KUKA KRL program: makrostep9.src

&ACCESS RVO
&COMMENT MakroStep9-Basic
&PARAM TEMPLATE = C:\KRC\Roboter\Template\makrostepvorgabe.src
&PARAM EDITMASK = MakroStep
&PARAM TPVW_VERSION = 8.3.15
DEF MAKROSTEP9(Function :IN)
   ; FOLD Makro Schrittkette;%{SE} %MKUKATPVW
   ; FOLD ;%{H} %MKUKATPVW
   INT Function
   IF Function==1 THEN
     APP_INT_STEP[9]=1
     Return
   ENDIF
   SWITCH APP_INT_STEP[9]
   Case 0
   ; ENDFOLD
   ;ENDFOLD
   ;FOLD SCHRITT 1 -- -- ;%{P}%MKUKATPVW,%CSTEP,%VST_NR,%P 1:SCHRITT, 2:1, 3:
      ;FOLD ;%{H}
         Case 1
      ;ENDFOLD
      ;FOLD -- Roboter Schrittkette -- ;%{SE}%MKUKATPVW %CVW_COM %VCOMMENT %P 2:-- Roboter Schrittkette --, 3: VW_COMMENT
      ;ENDFOLD
      ;FOLD -- KS26 -- ;%{SE}%MKUKATPVW %CVW_COM %VCOMMENT %P 2:-- KS26 --, 3: VW_COMMENT
      ;ENDFOLD
      ;FOLD -- Version: 01 -- ;%{SE}%MKUKATPVW %CVW_COM %VCOMMENT %P 2:-- Version: 01 --, 3: VW_COMMENT
      ;ENDFOLD
      ;FOLD -- Stand: 008 -- ;%{SE}%MKUKATPVW %CVW_COM %VCOMMENT %P 2:-- Stand: 008 --, 3: VW_COMMENT
      ;ENDFOLD
      ;FOLD -- letzte Aenderung 11.07.2019 LZ -- ;%{SE}%MKUKATPVW %CVW_COM %VCOMMENT %P 2:-- letzte Aenderung 11.07.2019 LZ --, 3: VW_COMMENT
      ;ENDFOLD
      ;FOLD -- E/A's und Flags Ruecksetzen -- ;%{SE}%MKUKATPVW %CVW_COM %VCOMMENT %P 2:-- E/A's und Flags Ruecksetzen --, 3: VW_COMMENT
      ;ENDFOLD
      ;FOLD -- SK1 KF1 KS1 KE1 -- ;%{SE}%MKUKATPVW %CVW_COM %VCOMMENT %P 2:-- SK1 KF1 KS1 KE1 --, 3: VW_COMMENT
      ;ENDFOLD
      ;FOLD A786 = F830 & A786 ;%{SE}%MKUKATPVW %CVW_SPS %VBOASG %P 2:A786 = F830 & A786, 3: BOASG
         $OUT[786] = $FLAG[830] AND $OUT[786]
      ;ENDFOLD
      ;FOLD A722 = !F830 & A722 ;%{SE}%MKUKATPVW %CVW_SPS %VBOASG %P 2:A722 = !F830 & A722, 3: BOASG
         $OUT[722] = NOT $FLAG[830] AND $OUT[722]
      ;ENDFOLD
      ;FOLD A834 = AUS ;%{SE}%MKUKATPVW %CVW_SPS %VBOASG %P 2:A834 = AUS, 3: BOASG
         $OUT[834] = FALSE
      ;ENDFOLD
      ;FOLD A840 = AUS ;%{SE}%MKUKATPVW %CVW_SPS %VBOASG %P 2:A840 = AUS, 3: BOASG
         $OUT[840] = FALSE
      ;ENDFOLD
      ;FOLD A757 = AUS ;%{SE}%MKUKATPVW %CVW_SPS %VBOASG %P 2:A757 = AUS, 3: BOASG
         $OUT[757] = FALSE
      ;ENDFOLD
      ;FOLD -- SK2 KF2 KS2 KE2 -- ;%{SE}%MKUKATPVW %CVW_COM %VCOMMENT %P 2:-- SK2 KF2 KS2 KE2 --, 3: VW_COMMENT
      ;ENDFOLD
      ;FOLD A946 = F831 & A946 ;%{SE}%MKUKATPVW %CVW_SPS %VBOASG %P 2:A946 = F831 & A946, 3: BOASG
         $OUT[946] = $FLAG[831] AND $OUT[946]
      ;ENDFOLD
      ;FOLD A882 = !F831 & A882 ;%{SE}%MKUKATPVW %CVW_SPS %VBOASG %P 2:A882 = !F831 & A882, 3: BOASG
         $OUT[882] = NOT $FLAG[831] AND $OUT[882]
      ;ENDFOLD
      ;FOLD A994 = AUS ;%{SE}%MKUKATPVW %CVW_SPS %VBOASG %P 2:A994 = AUS, 3: BOASG
         $OUT[994] = FALSE
      ;ENDFOLD
      ;FOLD A995 = AUS ;%{SE}%MKUKATPVW %CVW_SPS %VBOASG %P 2:A995 = AUS, 3: BOASG
         $OUT[995] = FALSE
      ;ENDFOLD
      ;FOLD A1000 = AUS ;%{SE}%MKUKATPVW %CVW_SPS %VBOASG %P 2:A1000 = AUS, 3: BOASG
         $OUT[1000] = FALSE
      ;ENDFOLD
      ;FOLD -- SK3 KF3 KS3 KE3 -- ;%{SE}%MKUKATPVW %CVW_COM %VCOMMENT %P 2:-- SK3 KF3 KS3 KE3 --, 3: VW_COMMENT
      ;ENDFOLD
      ;FOLD A1106 = F832 & A1106 ;%{SE}%MKUKATPVW %CVW_SPS %VBOASG %P 2:A1106 = F832 & A1106, 3: BOASG
         $OUT[1106] = $FLAG[832] AND $OUT[1106]
      ;ENDFOLD
      ;FOLD A1042 = !F832 & A1042 ;%{SE}%MKUKATPVW %CVW_SPS %VBOASG %P 2:A1042 = !F832 & A1042, 3: BOASG
         $OUT[1042] = NOT $FLAG[832] AND $OUT[1042]
      ;ENDFOLD
      ;FOLD A1154 = AUS ;%{SE}%MKUKATPVW %CVW_SPS %VBOASG %P 2:A1154 = AUS, 3: BOASG
         $OUT[1154] = FALSE
      ;ENDFOLD
      ;FOLD A1155 = AUS ;%{SE}%MKUKATPVW %CVW_SPS %VBOASG %P 2:A1155 = AUS, 3: BOASG
         $OUT[1155] = FALSE
      ;ENDFOLD
      ;FOLD A1160 = AUS ;%{SE}%MKUKATPVW %CVW_SPS %VBOASG %P 2:A1160 = AUS, 3: BOASG
         $OUT[1160] = FALSE
      ;ENDFOLD
      ;FOLD -- Auswertung KF Umdrehungen ServoGun -- ;%{SE}%MKUKATPVW %CVW_COM %VCOMMENT %P 2:-- Auswertung KF Umdrehungen ServoGun --, 3: VW_COMMENT
      ;ENDFOLD
      ;FOLD F94 = AUS ;%{SE}%MKUKATPVW %CVW_SPS %VBOASG %P 2:F94 = AUS, 3: BOASG
         $FLAG[94] = FALSE
      ;ENDFOLD
      ;FOLD F95 = AUS ;%{SE}%MKUKATPVW %CVW_SPS %VBOASG %P 2:F95 = AUS, 3: BOASG
         $FLAG[95] = FALSE
      ;ENDFOLD
      ;FOLD F96 = AUS ;%{SE}%MKUKATPVW %CVW_SPS %VBOASG %P 2:F96 = AUS, 3: BOASG
         $FLAG[96] = FALSE
      ;ENDFOLD
      ;FOLD F97 = AUS ;%{SE}%MKUKATPVW %CVW_SPS %VBOASG %P 2:F97 = AUS, 3: BOASG
         $FLAG[97] = FALSE
      ;ENDFOLD
      ;FOLD F98 = AUS ;%{SE}%MKUKATPVW %CVW_SPS %VBOASG %P 2:F98 = AUS, 3: BOASG
         $FLAG[98] = FALSE
      ;ENDFOLD
      ;FOLD F99 = AUS ;%{SE}%MKUKATPVW %CVW_SPS %VBOASG %P 2:F99 = AUS, 3: BOASG
         $FLAG[99] = FALSE
      ;ENDFOLD
      ;FOLD F100 = AUS ;%{SE}%MKUKATPVW %CVW_SPS %VBOASG %P 2:F100 = AUS, 3: BOASG
         $FLAG[100] = FALSE
      ;ENDFOLD
      ;FOLD F101 = AUS ;%{SE}%MKUKATPVW %CVW_SPS %VBOASG %P 2:F101 = AUS, 3: BOASG
         $FLAG[101] = FALSE
      ;ENDFOLD
      ;FOLD F102 = AUS ;%{SE}%MKUKATPVW %CVW_SPS %VBOASG %P 2:F102 = AUS, 3: BOASG
         $FLAG[102] = FALSE
      ;ENDFOLD
      ;FOLD F103 = AUS ;%{SE}%MKUKATPVW %CVW_SPS %VBOASG %P 2:F103 = AUS, 3: BOASG
         $FLAG[103] = FALSE
      ;ENDFOLD
      ;FOLD F104 = AUS ;%{SE}%MKUKATPVW %CVW_SPS %VBOASG %P 2:F104 = AUS, 3: BOASG
         $FLAG[104] = FALSE
      ;ENDFOLD
      ;FOLD F105 = AUS ;%{SE}%MKUKATPVW %CVW_SPS %VBOASG %P 2:F105 = AUS, 3: BOASG
         $FLAG[105] = FALSE
      ;ENDFOLD
      ;FOLD F106 = AUS ;%{SE}%MKUKATPVW %CVW_SPS %VBOASG %P 2:F106 = AUS, 3: BOASG
         $FLAG[106] = FALSE
      ;ENDFOLD
      ;FOLD F107 = AUS ;%{SE}%MKUKATPVW %CVW_SPS %VBOASG %P 2:F107 = AUS, 3: BOASG
         $FLAG[107] = FALSE
      ;ENDFOLD
      ;FOLD F108 = AUS ;%{SE}%MKUKATPVW %CVW_SPS %VBOASG %P 2:F108 = AUS, 3: BOASG
         $FLAG[108] = FALSE
      ;ENDFOLD
      ;FOLD F109 = AUS ;%{SE}%MKUKATPVW %CVW_SPS %VBOASG %P 2:F109 = AUS, 3: BOASG
         $FLAG[109] = FALSE
      ;ENDFOLD
      ;FOLD F110 = AUS ;%{SE}%MKUKATPVW %CVW_SPS %VBOASG %P 2:F110 = AUS, 3: BOASG
         $FLAG[110] = FALSE
      ;ENDFOLD
      ;FOLD F111 = AUS ;%{SE}%MKUKATPVW %CVW_SPS %VBOASG %P 2:F111 = AUS, 3: BOASG
         $FLAG[111] = FALSE
      ;ENDFOLD
      ;FOLD F112 = AUS ;%{SE}%MKUKATPVW %CVW_SPS %VBOASG %P 2:F112 = AUS, 3: BOASG
         $FLAG[112] = FALSE
      ;ENDFOLD
      ;FOLD F113 = AUS ;%{SE}%MKUKATPVW %CVW_SPS %VBOASG %P 2:F113 = AUS, 3: BOASG
         $FLAG[113] = FALSE
      ;ENDFOLD
      ;FOLD F114 = AUS ;%{SE}%MKUKATPVW %CVW_SPS %VBOASG %P 2:F114 = AUS, 3: BOASG
         $FLAG[114] = FALSE
      ;ENDFOLD
      ;FOLD F115 = AUS ;%{SE}%MKUKATPVW %CVW_SPS %VBOASG %P 2:F115 = AUS, 3: BOASG
         $FLAG[115] = FALSE
      ;ENDFOLD
      ;FOLD F116 = AUS ;%{SE}%MKUKATPVW %CVW_SPS %VBOASG %P 2:F116 = AUS, 3: BOASG
         $FLAG[116] = FALSE
      ;ENDFOLD
      ;FOLD F117 = AUS ;%{SE}%MKUKATPVW %CVW_SPS %VBOASG %P 2:F117 = AUS, 3: BOASG
         $FLAG[117] = FALSE
      ;ENDFOLD
      ;FOLD -- Auswertung KF Umdrehungen EZ2/SP2/KE2 -- ;%{SE}%MKUKATPVW %CVW_COM %VCOMMENT %P 2:-- Auswertung KF Umdrehungen EZ2/SP2/KE2 --, 3: VW_COMMENT
      ;ENDFOLD
      ;FOLD F150 = AUS ;%{SE}%MKUKATPVW %CVW_SPS %VBOASG %P 2:F150 = AUS, 3: BOASG
         $FLAG[150] = FALSE
      ;ENDFOLD
      ;FOLD F151 = AUS ;%{SE}%MKUKATPVW %CVW_SPS %VBOASG %P 2:F151 = AUS, 3: BOASG
         $FLAG[151] = FALSE
      ;ENDFOLD
      ;FOLD F152 = AUS ;%{SE}%MKUKATPVW %CVW_SPS %VBOASG %P 2:F152 = AUS, 3: BOASG
         $FLAG[152] = FALSE
      ;ENDFOLD
      ;FOLD F153 = AUS ;%{SE}%MKUKATPVW %CVW_SPS %VBOASG %P 2:F153 = AUS, 3: BOASG
         $FLAG[153] = FALSE
      ;ENDFOLD
      ;FOLD F154 = AUS ;%{SE}%MKUKATPVW %CVW_SPS %VBOASG %P 2:F154 = AUS, 3: BOASG
         $FLAG[154] = FALSE
      ;ENDFOLD
      ;FOLD F155 = AUS ;%{SE}%MKUKATPVW %CVW_SPS %VBOASG %P 2:F155 = AUS, 3: BOASG
         $FLAG[155] = FALSE
      ;ENDFOLD
      ;FOLD -- Auswertung KF Umdrehungen EZ3/SP3/KE3 -- ;%{SE}%MKUKATPVW %CVW_COM %VCOMMENT %P 2:-- Auswertung KF Umdrehungen EZ3/SP3/KE3 --, 3: VW_COMMENT
      ;ENDFOLD
      ;FOLD F186 = AUS ;%{SE}%MKUKATPVW %CVW_SPS %VBOASG %P 2:F186 = AUS, 3: BOASG
         $FLAG[186] = FALSE
      ;ENDFOLD
      ;FOLD F187 = AUS ;%{SE}%MKUKATPVW %CVW_SPS %VBOASG %P 2:F187 = AUS, 3: BOASG
         $FLAG[187] = FALSE
      ;ENDFOLD
      ;FOLD F188 = AUS ;%{SE}%MKUKATPVW %CVW_SPS %VBOASG %P 2:F188 = AUS, 3: BOASG
         $FLAG[188] = FALSE
      ;ENDFOLD
      ;FOLD F189 = AUS ;%{SE}%MKUKATPVW %CVW_SPS %VBOASG %P 2:F189 = AUS, 3: BOASG
         $FLAG[189] = FALSE
      ;ENDFOLD
      ;FOLD F190 = AUS ;%{SE}%MKUKATPVW %CVW_SPS %VBOASG %P 2:F190 = AUS, 3: BOASG
         $FLAG[190] = FALSE
      ;ENDFOLD
      ;FOLD F191 = AUS ;%{SE}%MKUKATPVW %CVW_SPS %VBOASG %P 2:F191 = AUS, 3: BOASG
         $FLAG[191] = FALSE
      ;ENDFOLD
      ;FOLD -- Hilfsflags beim Fraesen -- ;%{SE}%MKUKATPVW %CVW_COM %VCOMMENT %P 2:-- Hilfsflags beim Fraesen --, 3: VW_COMMENT
      ;ENDFOLD
      ;FOLD F749 = AUS ;%{SE}%MKUKATPVW %CVW_SPS %VBOASG %P 2:F749 = AUS, 3: BOASG
         $FLAG[749] = FALSE
      ;ENDFOLD
      ;FOLD F287 = AUS ;%{SE}%MKUKATPVW %CVW_SPS %VBOASG %P 2:F287 = AUS, 3: BOASG
         $FLAG[287] = FALSE
      ;ENDFOLD
      ;FOLD F290 = AUS ;%{SE}%MKUKATPVW %CVW_SPS %VBOASG %P 2:F290 = AUS, 3: BOASG
         $FLAG[290] = FALSE
      ;ENDFOLD
      ;FOLD F291 = AUS ;%{SE}%MKUKATPVW %CVW_SPS %VBOASG %P 2:F291 = AUS, 3: BOASG
         $FLAG[291] = FALSE
      ;ENDFOLD
      ;FOLD -- Hilfsflags SZ2 an SK1 -- ;%{SE}%MKUKATPVW %CVW_COM %VCOMMENT %P 2:-- Hilfsflags SZ2 an SK1 --, 3: VW_COMMENT
      ;ENDFOLD
      ;FOLD F307 = AUS ;%{SE}%MKUKATPVW %CVW_SPS %VBOASG %P 2:F307 = AUS, 3: BOASG
         $FLAG[307] = FALSE
      ;ENDFOLD
      ;FOLD F308 = AUS ;%{SE}%MKUKATPVW %CVW_SPS %VBOASG %P 2:F308 = AUS, 3: BOASG
         $FLAG[308] = FALSE
      ;ENDFOLD
      ;FOLD -- Hilfsflags Funktionstest KF Motor -- ;%{SE}%MKUKATPVW %CVW_COM %VCOMMENT %P 2:-- Hilfsflags Funktionstest KF Motor --, 3: VW_COMMENT
      ;ENDFOLD
      ;FOLD F312 = AUS ;%{SE}%MKUKATPVW %CVW_SPS %VBOASG %P 2:F312 = AUS, 3: BOASG
         $FLAG[312] = FALSE
      ;ENDFOLD
      ;FOLD F313 = AUS ;%{SE}%MKUKATPVW %CVW_SPS %VBOASG %P 2:F313 = AUS, 3: BOASG
         $FLAG[313] = FALSE
      ;ENDFOLD
      ;FOLD -- RSK Fehlerausgaben -- ;%{SE}%MKUKATPVW %CVW_COM %VCOMMENT %P 2:-- RSK Fehlerausgaben --, 3: VW_COMMENT
      ;ENDFOLD
      ;FOLD F322 = AUS ;%{SE}%MKUKATPVW %CVW_SPS %VBOASG %P 2:F322 = AUS, 3: BOASG
         $FLAG[322] = FALSE
      ;ENDFOLD
      ;FOLD F323 = AUS ;%{SE}%MKUKATPVW %CVW_SPS %VBOASG %P 2:F323 = AUS, 3: BOASG
         $FLAG[323] = FALSE
      ;ENDFOLD
      ;FOLD F324 = AUS ;%{SE}%MKUKATPVW %CVW_SPS %VBOASG %P 2:F324 = AUS, 3: BOASG
         $FLAG[324] = FALSE
      ;ENDFOLD
      ;FOLD F325 = AUS ;%{SE}%MKUKATPVW %CVW_SPS %VBOASG %P 2:F325 = AUS, 3: BOASG
         $FLAG[325] = FALSE
      ;ENDFOLD
      ;FOLD F326 = AUS ;%{SE}%MKUKATPVW %CVW_SPS %VBOASG %P 2:F326 = AUS, 3: BOASG
         $FLAG[326] = FALSE
      ;ENDFOLD
      ;FOLD F327 = AUS ;%{SE}%MKUKATPVW %CVW_SPS %VBOASG %P 2:F327 = AUS, 3: BOASG
         $FLAG[327] = FALSE
      ;ENDFOLD
      ;FOLD F328 = AUS ;%{SE}%MKUKATPVW %CVW_SPS %VBOASG %P 2:F328 = AUS, 3: BOASG
         $FLAG[328] = FALSE
      ;ENDFOLD
      ;FOLD F329 = AUS ;%{SE}%MKUKATPVW %CVW_SPS %VBOASG %P 2:F329 = AUS, 3: BOASG
         $FLAG[329] = FALSE
      ;ENDFOLD
      ;FOLD A3518 = AUS ;%{SE}%MKUKATPVW %CVW_SPS %VBOASG %P 2:A3518 = AUS, 3: BOASG
         $OUT[3518] = FALSE
      ;ENDFOLD
      ;FOLD A3519 = AUS ;%{SE}%MKUKATPVW %CVW_SPS %VBOASG %P 2:A3519 = AUS, 3: BOASG
         $OUT[3519] = FALSE
      ;ENDFOLD
      ;FOLD -- Schritt Fraesen aktiv -- ;%{SE}%MKUKATPVW %CVW_COM %VCOMMENT %P 2:-- Schritt Fraesen aktiv --, 3: VW_COMMENT
      ;ENDFOLD
      ;FOLD A3534 = AUS ;%{SE}%MKUKATPVW %CVW_SPS %VBOASG %P 2:A3534 = AUS, 3: BOASG
         $OUT[3534] = FALSE
      ;ENDFOLD
      ;FOLD -- Schritt Messen aktiv -- ;%{SE}%MKUKATPVW %CVW_COM %VCOMMENT %P 2:-- Schritt Messen aktiv --, 3: VW_COMMENT
      ;ENDFOLD
      ;FOLD A3535 = AUS ;%{SE}%MKUKATPVW %CVW_SPS %VBOASG %P 2:A3535 = AUS, 3: BOASG
         $OUT[3535] = FALSE
      ;ENDFOLD
      ;FOLD -- Schritt Schweissen aktiv -- ;%{SE}%MKUKATPVW %CVW_COM %VCOMMENT %P 2:-- Schritt Schweissen aktiv --, 3: VW_COMMENT
      ;ENDFOLD
      ;FOLD A3536 = AUS ;%{SE}%MKUKATPVW %CVW_SPS %VBOASG %P 2:A3536 = AUS, 3: BOASG
         $OUT[3536] = FALSE
      ;ENDFOLD
      ;FOLD -- Hilfsflag SK Programmwechsel -- ;%{SE}%MKUKATPVW %CVW_COM %VCOMMENT %P 2:-- Hilfsflag SK Programmwechsel --, 3: VW_COMMENT
      ;ENDFOLD
      ;FOLD F334 = AUS ;%{SE}%MKUKATPVW %CVW_SPS %VBOASG %P 2:F334 = AUS, 3: BOASG
         $FLAG[334] = FALSE
      ;ENDFOLD
      ;FOLD -- Timer Stoppen -- ;%{SE}%MKUKATPVW %CVW_COM %VCOMMENT %P 2:-- Timer Stoppen --, 3: VW_COMMENT
      ;ENDFOLD
      ;FOLD t7 ( EIN ) = STOP ;%{SE}%MKUKATPVW %CVW_SPS %VTSTOP %P 2:t7 ( EIN ) = STOP, 3: TSTOP
         VW(#SET_TIME,TRUE,7,1,0)
      ;ENDFOLD
      ;FOLD t8 ( EIN ) = STOP ;%{SE}%MKUKATPVW %CVW_SPS %VTSTOP %P 2:t8 ( EIN ) = STOP, 3: TSTOP
         VW(#SET_TIME,TRUE,8,1,0)
      ;ENDFOLD
      ;FOLD t9 ( EIN ) = STOP ;%{SE}%MKUKATPVW %CVW_SPS %VTSTOP %P 2:t9 ( EIN ) = STOP, 3: TSTOP
         VW(#SET_TIME,TRUE,9,1,0)
      ;ENDFOLD
      ;FOLD Schritt 2 = EIN ;%{SE}%MKUKATPVW %CVW_SPS %VST_CON %P 2:Schritt 2 = EIN, 3: ST_CON
         IF TRUE THEN
            PREV_STEP[9] = APP_INT_STEP[9]
            APP_INT_STEP[9] = 2
         ENDIF
      ;ENDFOLD
   ;ENDFOLD
   ;FOLD SCHRITT 2 --  RSK Grundstellung # Anwahlen-- ;%{P}%MKUKATPVW,%CSTEP,%VST_NR,%P 1:SCHRITT, 2:2, 3:  RSK Grundstellung # Anwahlen
      ;FOLD ;%{H}
         Case 2
      ;ENDFOLD
      ;FOLD -- RSK ServoZange in Grundstellung AUS -- ;%{SE}%MKUKATPVW %CVW_COM %VCOMMENT %P 2:-- RSK ServoZange in Grundstellung AUS --, 3: VW_COMMENT
      ;ENDFOLD
      ;FOLD F276 = AUS ;%{SE}%MKUKATPVW %CVW_SPS %VBOASG %P 2:F276 = AUS, 3: BOASG
         $FLAG[276] = FALSE
      ;ENDFOLD
      ;FOLD -- Fraesen st. RZ Start -- ;%{SE}%MKUKATPVW %CVW_COM %VCOMMENT %P 2:-- Fraesen st. RZ Start --, 3: VW_COMMENT
      ;ENDFOLD
      ;FOLD Schritt 103 = F92 & !F93 & A4039 & E13 & F273 & !F274 & !F275 & !F530 ;%{SE}%MKUKATPVW %CVW_SPS %VST_CON %P 2:Schritt 103 = F92 & !F93 & A4039 & E13 & F273 & !F274 & !F275 & !F530, 3: ST_CON
         IF $FLAG[92] AND NOT $FLAG[93] AND $OUT[4039] AND $IN[13] AND $FLAG[273] AND NOT $FLAG[274] AND NOT $FLAG[275] AND NOT $FLAG[530] THEN
            PREV_STEP[9] = APP_INT_STEP[9]
            APP_INT_STEP[9] = 103
         ENDIF
      ;ENDFOLD
      ;FOLD Schritt 203 = F148 & !F149 & A4039 & E13 & F273 & F274 & !F275  & !F530 ;%{SE}%MKUKATPVW %CVW_SPS %VST_CON %P 2:Schritt 203 = F148 & !F149 & A4039 & E13 & F273 & F274 & !F275  & !F530, 3: ST_CON
         IF $FLAG[148] AND NOT $FLAG[149] AND $OUT[4039] AND $IN[13] AND $FLAG[273] AND $FLAG[274] AND NOT $FLAG[275] AND NOT $FLAG[530] THEN
            PREV_STEP[9] = APP_INT_STEP[9]
            APP_INT_STEP[9] = 203
         ENDIF
      ;ENDFOLD
      ;FOLD Schritt 303 = F184 & !F185 & A4039 & E13 & F273 & F274 & F275  & !F530 ;%{SE}%MKUKATPVW %CVW_SPS %VST_CON %P 2:Schritt 303 = F184 & !F185 & A4039 & E13 & F273 & F274 & F275  & !F530, 3: ST_CON
         IF $FLAG[184] AND NOT $FLAG[185] AND $OUT[4039] AND $IN[13] AND $FLAG[273] AND $FLAG[274] AND $FLAG[275] AND NOT $FLAG[530] THEN
            PREV_STEP[9] = APP_INT_STEP[9]
            APP_INT_STEP[9] = 303
         ENDIF
      ;ENDFOLD
      ;FOLD Schritt 500 = A757 & A4039 & E13 & F273 & F530 ;%{SE}%MKUKATPVW %CVW_SPS %VST_CON %P 2:Schritt 500 = A757 & A4039 & E13 & F273 & F530, 3: ST_CON
         IF $OUT[757] AND $OUT[4039] AND $IN[13] AND $FLAG[273] AND $FLAG[530] THEN
            PREV_STEP[9] = APP_INT_STEP[9]
            APP_INT_STEP[9] = 500
         ENDIF
      ;ENDFOLD
   ;ENDFOLD
   ;FOLD SCHRITT 103 -- st. RZ1 # Start -- ;%{P}%MKUKATPVW,%CSTEP,%VST_NR,%P 1:SCHRITT, 2:103, 3: st. RZ1 # Start
      ;FOLD ;%{H}
         Case 103
      ;ENDFOLD
      ;FOLD -- RSK gestartet -- ;%{SE}%MKUKATPVW %CVW_COM %VCOMMENT %P 2:-- RSK gestartet --, 3: VW_COMMENT
      ;ENDFOLD
      ;FOLD F122 = AUS ;%{SE}%MKUKATPVW %CVW_SPS %VBOASG %P 2:F122 = AUS, 3: BOASG
         $FLAG[122] = FALSE
      ;ENDFOLD
      ;FOLD F322 = AUS ;%{SE}%MKUKATPVW %CVW_SPS %VBOASG %P 2:F322 = AUS, 3: BOASG
         $FLAG[322] = FALSE
      ;ENDFOLD
      ;FOLD F323 = AUS ;%{SE}%MKUKATPVW %CVW_SPS %VBOASG %P 2:F323 = AUS, 3: BOASG
         $FLAG[323] = FALSE
      ;ENDFOLD
      ;FOLD F324 = AUS ;%{SE}%MKUKATPVW %CVW_SPS %VBOASG %P 2:F324 = AUS, 3: BOASG
         $FLAG[324] = FALSE
      ;ENDFOLD
      ;FOLD F325 = AUS ;%{SE}%MKUKATPVW %CVW_SPS %VBOASG %P 2:F325 = AUS, 3: BOASG
         $FLAG[325] = FALSE
      ;ENDFOLD
      ;FOLD F326 = AUS ;%{SE}%MKUKATPVW %CVW_SPS %VBOASG %P 2:F326 = AUS, 3: BOASG
         $FLAG[326] = FALSE
      ;ENDFOLD
      ;FOLD F327 = AUS ;%{SE}%MKUKATPVW %CVW_SPS %VBOASG %P 2:F327 = AUS, 3: BOASG
         $FLAG[327] = FALSE
      ;ENDFOLD
      ;FOLD F329 = AUS ;%{SE}%MKUKATPVW %CVW_SPS %VBOASG %P 2:F329 = AUS, 3: BOASG
         $FLAG[329] = FALSE
      ;ENDFOLD
      ;FOLD -- ServoGun SZ1 Zaehler -- ;%{SE}%MKUKATPVW %CVW_COM %VCOMMENT %P 2:-- ServoGun SZ1 Zaehler --, 3: VW_COMMENT
      ;ENDFOLD
      ;FOLD F94 = AUS ;%{SE}%MKUKATPVW %CVW_SPS %VBOASG %P 2:F94 = AUS, 3: BOASG
         $FLAG[94] = FALSE
      ;ENDFOLD
      ;FOLD F95 = AUS ;%{SE}%MKUKATPVW %CVW_SPS %VBOASG %P 2:F95 = AUS, 3: BOASG
         $FLAG[95] = FALSE
      ;ENDFOLD
      ;FOLD F96 = AUS ;%{SE}%MKUKATPVW %CVW_SPS %VBOASG %P 2:F96 = AUS, 3: BOASG
         $FLAG[96] = FALSE
      ;ENDFOLD
      ;FOLD F97 = AUS ;%{SE}%MKUKATPVW %CVW_SPS %VBOASG %P 2:F97 = AUS, 3: BOASG
         $FLAG[97] = FALSE
      ;ENDFOLD
      ;FOLD F98 = AUS ;%{SE}%MKUKATPVW %CVW_SPS %VBOASG %P 2:F98 = AUS, 3: BOASG
         $FLAG[98] = FALSE
      ;ENDFOLD
      ;FOLD F99 = AUS ;%{SE}%MKUKATPVW %CVW_SPS %VBOASG %P 2:F99 = AUS, 3: BOASG
         $FLAG[99] = FALSE
      ;ENDFOLD
      ;FOLD -- Hilfsflags Funktionstest KF Motor -- ;%{SE}%MKUKATPVW %CVW_COM %VCOMMENT %P 2:-- Hilfsflags Funktionstest KF Motor --, 3: VW_COMMENT
      ;ENDFOLD
      ;FOLD F312 = AUS ;%{SE}%MKUKATPVW %CVW_SPS %VBOASG %P 2:F312 = AUS, 3: BOASG
         $FLAG[312] = FALSE
      ;ENDFOLD
      ;FOLD F313 = AUS ;%{SE}%MKUKATPVW %CVW_SPS %VBOASG %P 2:F313 = AUS, 3: BOASG
         $FLAG[313] = FALSE
      ;ENDFOLD
      ;FOLD -- Hilfsflags ServoGun Start -- ;%{SE}%MKUKATPVW %CVW_COM %VCOMMENT %P 2:-- Hilfsflags ServoGun Start --, 3: VW_COMMENT
      ;ENDFOLD
      ;FOLD F276 = EIN ;%{SE}%MKUKATPVW %CVW_SPS %VBOASG %P 2:F276 = EIN, 3: BOASG
         $FLAG[276] = TRUE
      ;ENDFOLD
      ;FOLD A3871 = AUS ;%{SE}%MKUKATPVW %CVW_SPS %VBOASG %P 2:A3871 = AUS, 3: BOASG
         $OUT[3871] = FALSE
      ;ENDFOLD
      ;FOLD A3872 = AUS ;%{SE}%MKUKATPVW %CVW_SPS %VBOASG %P 2:A3872 = AUS, 3: BOASG
         $OUT[3872] = FALSE
      ;ENDFOLD
      ;FOLD A3510 = EIN ;%{SE}%MKUKATPVW %CVW_SPS %VBOASG %P 2:A3510 = EIN, 3: BOASG
         $OUT[3510] = TRUE
      ;ENDFOLD
      ;FOLD A3511 = AUS ;%{SE}%MKUKATPVW %CVW_SPS %VBOASG %P 2:A3511 = AUS, 3: BOASG
         $OUT[3511] = FALSE
      ;ENDFOLD
      ;FOLD A3514 = AUS ;%{SE}%MKUKATPVW %CVW_SPS %VBOASG %P 2:A3514 = AUS, 3: BOASG
         $OUT[3514] = FALSE
      ;ENDFOLD
      ;FOLD A3513 = AUS ;%{SE}%MKUKATPVW %CVW_SPS %VBOASG %P 2:A3513 = AUS, 3: BOASG
         $OUT[3513] = FALSE
      ;ENDFOLD
      ;FOLD A3512 = AUS ;%{SE}%MKUKATPVW %CVW_SPS %VBOASG %P 2:A3512 = AUS, 3: BOASG
         $OUT[3512] = FALSE
      ;ENDFOLD
      ;FOLD A3533 = AUS ;%{SE}%MKUKATPVW %CVW_SPS %VBOASG %P 2:A3533 = AUS, 3: BOASG
         $OUT[3533] = FALSE
      ;ENDFOLD
      ;FOLD A3534 = AUS ;%{SE}%MKUKATPVW %CVW_SPS %VBOASG %P 2:A3534 = AUS, 3: BOASG
         $OUT[3534] = FALSE
      ;ENDFOLD
      ;FOLD A3535 = AUS ;%{SE}%MKUKATPVW %CVW_SPS %VBOASG %P 2:A3535 = AUS, 3: BOASG
         $OUT[3535] = FALSE
      ;ENDFOLD
      ;FOLD A3536 = AUS ;%{SE}%MKUKATPVW %CVW_SPS %VBOASG %P 2:A3536 = AUS, 3: BOASG
         $OUT[3536] = FALSE
      ;ENDFOLD
      ;FOLD -- Hilfsflags ServoGun Ende -- ;%{SE}%MKUKATPVW %CVW_COM %VCOMMENT %P 2:-- Hilfsflags ServoGun Ende --, 3: VW_COMMENT
      ;ENDFOLD
      ;FOLD -- Ausblasen zuruecksetzen -- ;%{SE}%MKUKATPVW %CVW_COM %VCOMMENT %P 2:-- Ausblasen zuruecksetzen --, 3: VW_COMMENT
      ;ENDFOLD
      ;FOLD A836 = AUS ;%{SE}%MKUKATPVW %CVW_SPS %VBOASG %P 2:A836 = AUS, 3: BOASG
         $OUT[836] = FALSE
      ;ENDFOLD
      ;FOLD A996 = AUS ;%{SE}%MKUKATPVW %CVW_SPS %VBOASG %P 2:A996 = AUS, 3: BOASG
         $OUT[996] = FALSE
      ;ENDFOLD
      ;FOLD A1156 = AUS ;%{SE}%MKUKATPVW %CVW_SPS %VBOASG %P 2:A1156 = AUS, 3: BOASG
         $OUT[1156] = FALSE
      ;ENDFOLD
      ;FOLD -- Prognummer setzen -- ;%{SE}%MKUKATPVW %CVW_COM %VCOMMENT %P 2:-- Prognummer setzen --, 3: VW_COMMENT
      ;ENDFOLD
      ;FOLD bin28 ( EIN ) = 0 ;%{SE}%MKUKATPVW %CVW_SPS %VARIASG %P 2:bin28 ( EIN ) = 0, 3: ARIASG
         VW(#BINOUT,TRUE,28,0)
      ;ENDFOLD
      ;FOLD bin1 ( EIN ) = 31 ;%{SE}%MKUKATPVW %CVW_SPS %VARIASG %P 2:bin1 ( EIN ) = 31, 3: ARIASG
         VW(#BINOUT,TRUE,1,31)
      ;ENDFOLD
      ;FOLD bin30 ( EIN ) = p111 ;%{SE}%MKUKATPVW %CVW_SPS %VARIASG %P 2:bin30 ( EIN ) = p111, 3: ARIASG
         VW(#BINOUT,TRUE,30,PROCPAR[111])
      ;ENDFOLD
      ;FOLD bin31 ( EIN ) = 31 ;%{SE}%MKUKATPVW %CVW_SPS %VARIASG %P 2:bin31 ( EIN ) = 31, 3: ARIASG
         VW(#BINOUT,TRUE,31,31)
      ;ENDFOLD
      ;FOLD -- Wartezeit Programmwechsel SK -- ;%{SE}%MKUKATPVW %CVW_COM %VCOMMENT %P 2:-- Wartezeit Programmwechsel SK --, 3: VW_COMMENT
      ;ENDFOLD
      ;FOLD T8 ( !F334 ) = -2[1/10Sek] ;%{SE}%MKUKATPVW %CVW_SPS %VTASG %P 2:T8 ( !F334 ) = -2[1/10Sek], 3: TASG
         VW(#SET_TIME,NOT $FLAG[334],8,0,-2)
      ;ENDFOLD
      ;FOLD -- Hilfsflag SK Programmwechsel -- ;%{SE}%MKUKATPVW %CVW_COM %VCOMMENT %P 2:-- Hilfsflag SK Programmwechsel --, 3: VW_COMMENT
      ;ENDFOLD
      ;FOLD F334 = EIN ;%{SE}%MKUKATPVW %CVW_SPS %VBOASG %P 2:F334 = EIN, 3: BOASG
         $FLAG[334] = TRUE
      ;ENDFOLD
      ;FOLD -- Stat. ServoGun SZ1 beim Fraesen -- ;%{SE}%MKUKATPVW %CVW_COM %VCOMMENT %P 2:-- Stat. ServoGun SZ1 beim Fraesen --, 3: VW_COMMENT
      ;ENDFOLD
      ;FOLD A116 = EIN ;%{SE}%MKUKATPVW %CVW_SPS %VBOASG %P 2:A116 = EIN, 3: BOASG
         $OUT[116] = TRUE
      ;ENDFOLD
      ;FOLD A130 = EIN ;%{SE}%MKUKATPVW %CVW_SPS %VBOASG %P 2:A130 = EIN, 3: BOASG
         $OUT[130] = TRUE
      ;ENDFOLD
      ;FOLD -- Schritt Fraesen aktiv -- ;%{SE}%MKUKATPVW %CVW_COM %VCOMMENT %P 2:-- Schritt Fraesen aktiv --, 3: VW_COMMENT
      ;ENDFOLD
      ;FOLD A3534 = EIN ;%{SE}%MKUKATPVW %CVW_SPS %VBOASG %P 2:A3534 = EIN, 3: BOASG
         $OUT[3534] = TRUE
      ;ENDFOLD
      ;FOLD -- Quitt. Fraesen SK1 AUS -- ;%{SE}%MKUKATPVW %CVW_COM %VCOMMENT %P 2:-- Quitt. Fraesen SK1 AUS --, 3: VW_COMMENT
      ;ENDFOLD
      ;FOLD A786 = F830 ;%{SE}%MKUKATPVW %CVW_SPS %VBOASG %P 2:A786 = F830, 3: BOASG
         $OUT[786] = $FLAG[830]
      ;ENDFOLD
      ;FOLD A722 = !F830 ;%{SE}%MKUKATPVW %CVW_SPS %VBOASG %P 2:A722 = !F830, 3: BOASG
         $OUT[722] = NOT $FLAG[830]
      ;ENDFOLD
      ;FOLD Schritt 104 = A4039 ;%{SE}%MKUKATPVW %CVW_SPS %VST_CON %P 2:Schritt 104 = A4039, 3: ST_CON
         IF $OUT[4039] THEN
            PREV_STEP[9] = APP_INT_STEP[9]
            APP_INT_STEP[9] = 104
         ENDIF
      ;ENDFOLD
   ;ENDFOLD
   ;FOLD SCHRITT 104 -- st. RZ1 -- ;%{P}%MKUKATPVW,%CSTEP,%VST_NR,%P 1:SCHRITT, 2:104, 3: st. RZ1
      ;FOLD ;%{H}
         Case 104
      ;ENDFOLD
      ;FOLD -- Hilfsflag SK Programmwechsel -- ;%{SE}%MKUKATPVW %CVW_COM %VCOMMENT %P 2:-- Hilfsflag SK Programmwechsel --, 3: VW_COMMENT
      ;ENDFOLD
      ;FOLD F334 = AUS ;%{SE}%MKUKATPVW %CVW_SPS %VBOASG %P 2:F334 = AUS, 3: BOASG
         $FLAG[334] = FALSE
      ;ENDFOLD
      ;FOLD -- Wiederholfraesen aktiv -- ;%{SE}%MKUKATPVW %CVW_COM %VCOMMENT %P 2:-- Wiederholfraesen aktiv --, 3: VW_COMMENT
      ;ENDFOLD
      ;FOLD F327 = A3519 ;%{SE}%MKUKATPVW %CVW_SPS %VBOASG %P 2:F327 = A3519, 3: BOASG
         $FLAG[327] = $OUT[3519]
      ;ENDFOLD
      ;FOLD F749 = A3519 ;%{SE}%MKUKATPVW %CVW_SPS %VBOASG %P 2:F749 = A3519, 3: BOASG
         $FLAG[749] = $OUT[3519]
      ;ENDFOLD
      ;FOLD A144 = AUS ;%{SE}%MKUKATPVW %CVW_SPS %VBOASG %P 2:A144 = AUS, 3: BOASG
         $OUT[144] = FALSE
      ;ENDFOLD
      ;FOLD -- Ueberwachungszeit KF1 EIN -- ;%{SE}%MKUKATPVW %CVW_COM %VCOMMENT %P 2:-- Ueberwachungszeit KF1 EIN --, 3: VW_COMMENT
      ;ENDFOLD
      ;FOLD T7 ( EIN ) = -50[1/10Sek] ;%{SE}%MKUKATPVW %CVW_SPS %VTASG %P 2:T7 ( EIN ) = -50[1/10Sek], 3: TASG
         VW(#SET_TIME,TRUE,7,0,-50)
      ;ENDFOLD
      ;FOLD -- KF1 einschalten -- ;%{SE}%MKUKATPVW %CVW_COM %VCOMMENT %P 2:-- KF1 einschalten --, 3: VW_COMMENT
      ;ENDFOLD
      ;FOLD i1 (EIN) = 0 ;%{SE}%MKUKATPVW %CVW_SPS %VARIASG %P 2:i1 (EIN) = 0, 3: ARIASG
         VW(#COUNTER,TRUE,1,0)
      ;ENDFOLD
      ;FOLD A834 = EIN ;%{SE}%MKUKATPVW %CVW_SPS %VBOASG %P 2:A834 = EIN, 3: BOASG
         $OUT[834] = TRUE
      ;ENDFOLD
      ;FOLD SCHRITT 105 = A4039 ;%{SE}%MKUKATPVW %CVW_SPS %VST_CON %P 2:SCHRITT 105 = A4039, 3: ST_CON
         IF $OUT[4039] THEN
            PREV_STEP[9] = APP_INT_STEP[9]
            APP_INT_STEP[9] = 105
         ENDIF
      ;ENDFOLD
   ;ENDFOLD
   ;FOLD SCHRITT 105 -- st. RZ1 # Funktionstest KF -- ;%{P}%MKUKATPVW,%CSTEP,%VST_NR,%P 1:SCHRITT, 2:105, 3: st. RZ1 # Funktionstest KF
      ;FOLD ;%{H}
         Case 105
      ;ENDFOLD
      ;FOLD -- Funktionstest KF Motor -- ;%{SE}%MKUKATPVW %CVW_COM %VCOMMENT %P 2:-- Funktionstest KF Motor --, 3: VW_COMMENT
      ;ENDFOLD
      ;FOLD F312 = EIN ;%{SE}%MKUKATPVW %CVW_SPS %VBOASG %P 2:F312 = EIN, 3: BOASG
         $FLAG[312] = TRUE
      ;ENDFOLD
      ;FOLD F313 = i1 > 2 ;%{SE}%MKUKATPVW %CVW_SPS %VBOCMP %P 2:F313 = i1 > 2, 3: BOCMP
         $FLAG[313] = $COUNT_I[1] > 2
      ;ENDFOLD
      ;FOLD -- Ueberwachungszeit KS1 schwenken -- ;%{SE}%MKUKATPVW %CVW_COM %VCOMMENT %P 2:-- Ueberwachungszeit KS1 schwenken --, 3: VW_COMMENT
      ;ENDFOLD
      ;FOLD t8 ( EIN ) = -100[1/10Sek] ;%{SE}%MKUKATPVW %CVW_SPS %VTASG %P 2:t8 ( EIN ) = -100[1/10Sek], 3: TASG
         VW(#SET_TIME,TRUE,8,0,-100)
      ;ENDFOLD
      ;FOLD Schritt 107 = (F313 + T7) & A4039 ;%{SE}%MKUKATPVW %CVW_SPS %VST_CON %P 2:Schritt 107 = (F313 + T7) & A4039, 3: ST_CON
         IF ($FLAG[313] OR $TIMER_FLAG[7]) AND $OUT[4039] THEN
            PREV_STEP[9] = APP_INT_STEP[9]
            APP_INT_STEP[9] = 107
         ENDIF
      ;ENDFOLD
   ;ENDFOLD
   ;FOLD SCHRITT 107 -- st. RZ1 # Fehler KF -- ;%{P}%MKUKATPVW,%CSTEP,%VST_NR,%P 1:SCHRITT, 2:107, 3: st. RZ1 # Fehler KF
      ;FOLD ;%{H}
         Case 107
      ;ENDFOLD
      ;FOLD -- RSK Fehlerausgabe KF1 Initiator/Motor -- ;%{SE}%MKUKATPVW %CVW_COM %VCOMMENT %P 2:-- RSK Fehlerausgabe KF1 Initiator/Motor --, 3: VW_COMMENT
      ;ENDFOLD
      ;FOLD F322 = !F313 ;%{SE}%MKUKATPVW %CVW_SPS %VBOASG %P 2:F322 = !F313, 3: BOASG
         $FLAG[322] = NOT $FLAG[313]
      ;ENDFOLD
      ;FOLD -- RSK Fehlerausgabe KS1 Ruhest. -- ;%{SE}%MKUKATPVW %CVW_COM %VCOMMENT %P 2:-- RSK Fehlerausgabe KS1 Ruhest. --, 3: VW_COMMENT
      ;ENDFOLD
      ;FOLD F323 = (!E836 + E837 + E838 + !E839) & !F324 & !F328 ;%{SE}%MKUKATPVW %CVW_SPS %VBOASG %P 2:F323 = (!E836 + E837 + E838 + !E839) & !F324 & !F328, 3: BOASG
         $FLAG[323] = (NOT $IN[836] OR $IN[837] OR $IN[838] OR NOT $IN[839]) AND NOT $FLAG[324] AND NOT $FLAG[328]
      ;ENDFOLD
      ;FOLD -- RSK Sammelstoerung -- ;%{SE}%MKUKATPVW %CVW_COM %VCOMMENT %P 2:-- RSK Sammelstoerung --, 3: VW_COMMENT
      ;ENDFOLD
      ;FOLD F329 = F322 + F323 + T8 ;%{SE}%MKUKATPVW %CVW_SPS %VBOASG %P 2:F329 = F322 + F323 + T8, 3: BOASG
         $FLAG[329] = $FLAG[322] OR $FLAG[323] OR $TIMER_FLAG[8]
      ;ENDFOLD
      ;FOLD T7 ( EIN ) = STOP ;%{SE}%MKUKATPVW %CVW_SPS %VTSTOP %P 2:T7 ( EIN ) = STOP, 3: TSTOP
         VW(#SET_TIME,TRUE,7,1,0)
      ;ENDFOLD
      ;FOLD -- KF Motor Ein -- ;%{SE}%MKUKATPVW %CVW_COM %VCOMMENT %P 2:-- KF Motor Ein --, 3: VW_COMMENT
      ;ENDFOLD
      ;FOLD A834 = !F322 & !F323 ;%{SE}%MKUKATPVW %CVW_SPS %VBOASG %P 2:A834 = !F322 & !F323, 3: BOASG
         $OUT[834] = NOT $FLAG[322] AND NOT $FLAG[323]
      ;ENDFOLD
      ;FOLD -- KF1 Versetzeinheit vor -- ;%{SE}%MKUKATPVW %CVW_COM %VCOMMENT %P 2:-- KF1 Versetzeinheit vor --, 3: VW_COMMENT
      ;ENDFOLD
      ;FOLD A835 = !F322 & !F323 & F564 ;%{SE}%MKUKATPVW %CVW_SPS %VBOASG %P 2:A835 = !F322 & !F323 & F564, 3: BOASG
         $OUT[835] = NOT $FLAG[322] AND NOT $FLAG[323] AND $FLAG[564]
      ;ENDFOLD
      ;FOLD SCHRITT 108 = (!F322 & !F323) & (E835 & F564 + !E835 & !F564) & A4039 ;%{SE}%MKUKATPVW %CVW_SPS %VST_CON %P 2:SCHRITT 108 = (!F322 & !F323) & (E835 & F564 + !E835 & !F564) & A4039, 3: ST_CON
         IF (NOT $FLAG[322] AND NOT $FLAG[323]) AND ($IN[835] AND $FLAG[564] OR NOT $IN[835] AND NOT $FLAG[564]) AND $OUT[4039] THEN
            PREV_STEP[9] = APP_INT_STEP[9]
            APP_INT_STEP[9] = 108
         ENDIF
      ;ENDFOLD
      ;FOLD SCHRITT 134 = (F322 + F323) & !F324 & !F328 & A4039 & (E26 + E27) ;%{SE}%MKUKATPVW %CVW_SPS %VST_CON %P 2:SCHRITT 134 = (F322 + F323) & !F324 & !F328 & A4039 & (E26 + E27), 3: ST_CON
         IF ($FLAG[322] OR $FLAG[323]) AND NOT $FLAG[324] AND NOT $FLAG[328] AND $OUT[4039] AND ($IN[26] OR $IN[27]) THEN
            PREV_STEP[9] = APP_INT_STEP[9]
            APP_INT_STEP[9] = 134
         ENDIF
      ;ENDFOLD
   ;ENDFOLD
   ;FOLD SCHRITT 108 -- st. RZ1 # Sicherheit KF -- ;%{P}%MKUKATPVW,%CSTEP,%VST_NR,%P 1:SCHRITT, 2:108, 3: st. RZ1 # Sicherheit KF
      ;FOLD ;%{H}
         Case 108
      ;ENDFOLD
      ;FOLD -- RSK Sammelstoerung -- ;%{SE}%MKUKATPVW %CVW_COM %VCOMMENT %P 2:-- RSK Sammelstoerung --, 3: VW_COMMENT
      ;ENDFOLD
      ;FOLD F329 = AUS ;%{SE}%MKUKATPVW %CVW_SPS %VBOASG %P 2:F329 = AUS, 3: BOASG
         $FLAG[329] = FALSE
      ;ENDFOLD
      ;FOLD F324 = AUS ;%{SE}%MKUKATPVW %CVW_SPS %VBOASG %P 2:F324 = AUS, 3: BOASG
         $FLAG[324] = FALSE
      ;ENDFOLD
      ;FOLD F328 = AUS ;%{SE}%MKUKATPVW %CVW_SPS %VBOASG %P 2:F328 = AUS, 3: BOASG
         $FLAG[328] = FALSE
      ;ENDFOLD
      ;FOLD -- Wartebedingung schwenken -- ;%{SE}%MKUKATPVW %CVW_COM %VCOMMENT %P 2:-- Wartebedingung schwenken --, 3: VW_COMMENT
      ;ENDFOLD
      ;FOLD SCHRITT 109 = A3862 & A4039 ;%{SE}%MKUKATPVW %CVW_SPS %VST_CON %P 2:SCHRITT 109 = A3862 & A4039, 3: ST_CON
         IF $OUT[3862] AND $OUT[4039] THEN
            PREV_STEP[9] = APP_INT_STEP[9]
            APP_INT_STEP[9] = 109
         ENDIF
      ;ENDFOLD
   ;ENDFOLD
   ;FOLD SCHRITT 109 -- st. RZ1 # KS in AS schwenken -- ;%{P}%MKUKATPVW,%CSTEP,%VST_NR,%P 1:SCHRITT, 2:109, 3: st. RZ1 # KS in AS schwenken
      ;FOLD ;%{H}
         Case 109
      ;ENDFOLD
      ;FOLD -- KS1 in Arbeitsstellung schwenken -- ;%{SE}%MKUKATPVW %CVW_COM %VCOMMENT %P 2:-- KS1 in Arbeitsstellung schwenken --, 3: VW_COMMENT
      ;ENDFOLD
      ;FOLD A840 = A3862 & !E837 & (E835 & F564 + !E835 & !F564) ;%{SE}%MKUKATPVW %CVW_SPS %VBOASG %P 2:A840 = A3862 & !E837 & (E835 & F564 + !E835 & !F564), 3: BOASG
         $OUT[840] = $OUT[3862] AND NOT $IN[837] AND ($IN[835] AND $FLAG[564] OR NOT $IN[835] AND NOT $FLAG[564])
      ;ENDFOLD
      ;FOLD -- KF1 Ausblasen -- ;%{SE}%MKUKATPVW %CVW_COM %VCOMMENT %P 2:-- KF1 Ausblasen --, 3: VW_COMMENT
      ;ENDFOLD
      ;FOLD A836 = F330 + !F330 & !F331 & !F332 ;%{SE}%MKUKATPVW %CVW_SPS %VBOASG %P 2:A836 = F330 + !F330 & !F331 & !F332, 3: BOASG
         $OUT[836] = $FLAG[330] OR NOT $FLAG[330] AND NOT $FLAG[331] AND NOT $FLAG[332]
      ;ENDFOLD
      ;FOLD SCHRITT 110 =  A3862 & (A840 + E837 + T8) & A4039 ;%{SE}%MKUKATPVW %CVW_SPS %VST_CON %P 2:SCHRITT 110 =  A3862 & (A840 + E837 + T8) & A4039, 3: ST_CON
         IF $OUT[3862] AND ($OUT[840] OR $IN[837] OR $TIMER_FLAG[8]) AND $OUT[4039] THEN
            PREV_STEP[9] = APP_INT_STEP[9]
            APP_INT_STEP[9] = 110
         ENDIF
      ;ENDFOLD
   ;ENDFOLD
   ;FOLD SCHRITT 110 -- st. RZ1 -- ;%{P}%MKUKATPVW,%CSTEP,%VST_NR,%P 1:SCHRITT, 2:110, 3: st. RZ1
      ;FOLD ;%{H}
         Case 110
      ;ENDFOLD
      ;FOLD -- RSK Fehlerausgabe KF Versetzeinheit -- ;%{SE}%MKUKATPVW %CVW_COM %VCOMMENT %P 2:-- RSK Fehlerausgabe KF Versetzeinheit --, 3: VW_COMMENT
      ;ENDFOLD
      ;FOLD F328 = !E835 & F564 & !F324 ;%{SE}%MKUKATPVW %CVW_SPS %VBOASG %P 2:F328 = !E835 & F564 & !F324, 3: BOASG
         $FLAG[328] = NOT $IN[835] AND $FLAG[564] AND NOT $FLAG[324]
      ;ENDFOLD
      ;FOLD -- RSK Fehlerausgabe KS1 Arbeitsstellung -- ;%{SE}%MKUKATPVW %CVW_COM %VCOMMENT %P 2:-- RSK Fehlerausgabe KS1 Arbeitsstellung --, 3: VW_COMMENT
      ;ENDFOLD
      ;FOLD F324 = (E836 + !E837 + !E838 + E839) & T8 & (E835 + !F564) + F324 ;%{SE}%MKUKATPVW %CVW_SPS %VBOASG %P 2:F324 = (E836 + !E837 + !E838 + E839) & T8 & (E835 + !F564) + F324, 3: BOASG
         $FLAG[324] = ($IN[836] OR NOT $IN[837] OR NOT $IN[838] OR $IN[839]) AND $TIMER_FLAG[8] AND ($IN[835] OR NOT $FLAG[564]) OR $FLAG[324]
      ;ENDFOLD
      ;FOLD -- RSK Fehlerausgabe EZ/SP min. Oeffnung -- ;%{SE}%MKUKATPVW %CVW_COM %VCOMMENT %P 2:-- RSK Fehlerausgabe EZ/SP min. Oeffnung --, 3: VW_COMMENT
      ;ENDFOLD
      ;FOLD F333 = !A3862 ;%{SE}%MKUKATPVW %CVW_SPS %VBOASG %P 2:F333 = !A3862, 3: BOASG
         $FLAG[333] = NOT $OUT[3862]
      ;ENDFOLD
      ;FOLD -- RSK Sammelstoerung -- ;%{SE}%MKUKATPVW %CVW_COM %VCOMMENT %P 2:-- RSK Sammelstoerung --, 3: VW_COMMENT
      ;ENDFOLD
      ;FOLD F329 = F324 + F328 + F333 ;%{SE}%MKUKATPVW %CVW_SPS %VBOASG %P 2:F329 = F324 + F328 + F333, 3: BOASG
         $FLAG[329] = $FLAG[324] OR $FLAG[328] OR $FLAG[333]
      ;ENDFOLD
      ;FOLD A834 = !F324 & !F328 ;%{SE}%MKUKATPVW %CVW_SPS %VBOASG %P 2:A834 = !F324 & !F328, 3: BOASG
         $OUT[834] = NOT $FLAG[324] AND NOT $FLAG[328]
      ;ENDFOLD
      ;FOLD -- Verweilzeit Versetzeinheit Rueck -- ;%{SE}%MKUKATPVW %CVW_COM %VCOMMENT %P 2:-- Verweilzeit Versetzeinheit Rueck --, 3: VW_COMMENT
      ;ENDFOLD
      ;FOLD t11 ( EIN ) = i24[1/10Sek] ;%{SE}%MKUKATPVW %CVW_SPS %VTASG %P 2:t11 ( EIN ) = i24[1/10Sek], 3: TASG
         VW(#SET_TIME,TRUE,11,0,$COUNT_I[24])
      ;ENDFOLD
      ;FOLD -- KF1 Ausblasen -- ;%{SE}%MKUKATPVW %CVW_COM %VCOMMENT %P 2:-- KF1 Ausblasen --, 3: VW_COMMENT
      ;ENDFOLD
      ;FOLD A836 = (F330 + !F330 & !F331 & !F332) & !F324 & !F328 ;%{SE}%MKUKATPVW %CVW_SPS %VBOASG %P 2:A836 = (F330 + !F330 & !F331 & !F332) & !F324 & !F328, 3: BOASG
         $OUT[836] = ($FLAG[330] OR NOT $FLAG[330] AND NOT $FLAG[331] AND NOT $FLAG[332]) AND NOT $FLAG[324] AND NOT $FLAG[328]
      ;ENDFOLD
      ;FOLD A835 = F564 ;%{SE}%MKUKATPVW %CVW_SPS %VBOASG %P 2:A835 = F564, 3: BOASG
         $OUT[835] = $FLAG[564]
      ;ENDFOLD
      ;FOLD Schritt 103 = (F324 + F328) & (E26 + E27) & A4039 ;%{SE}%MKUKATPVW %CVW_SPS %VST_CON %P 2:Schritt 103 = (F324 + F328) & (E26 + E27) & A4039, 3: ST_CON
         IF ($FLAG[324] OR $FLAG[328]) AND ($IN[26] OR $IN[27]) AND $OUT[4039] THEN
            PREV_STEP[9] = APP_INT_STEP[9]
            APP_INT_STEP[9] = 103
         ENDIF
      ;ENDFOLD
      ;FOLD SCHRITT 111 = !F324 & !F328 & !E836 & E837 & E838 & !E839 & A4039 ;%{SE}%MKUKATPVW %CVW_SPS %VST_CON %P 2:SCHRITT 111 = !F324 & !F328 & !E836 & E837 & E838 & !E839 & A4039, 3: ST_CON
         IF NOT $FLAG[324] AND NOT $FLAG[328] AND NOT $IN[836] AND $IN[837] AND $IN[838] AND NOT $IN[839] AND $OUT[4039] THEN
            PREV_STEP[9] = APP_INT_STEP[9]
            APP_INT_STEP[9] = 111
         ENDIF
      ;ENDFOLD
   ;ENDFOLD
   ;FOLD SCHRITT 111 -- st. RZ1 -- ;%{P}%MKUKATPVW,%CSTEP,%VST_NR,%P 1:SCHRITT, 2:111, 3: st. RZ1
      ;FOLD ;%{H}
         Case 111
      ;ENDFOLD
      ;FOLD -- Umdreh. KF setzen zwischenspeichern -- ;%{SE}%MKUKATPVW %CVW_COM %VCOMMENT %P 2:-- Umdreh. KF setzen zwischenspeichern --, 3: VW_COMMENT
      ;ENDFOLD
      ;FOLD i45 ( EIN ) = i4 ;%{SE}%MKUKATPVW %CVW_SPS %VARIASG %P 2:i45 ( EIN ) = i4, 3: ARIASG
         VW(#COUNTER,TRUE,45,$COUNT_I[4])
      ;ENDFOLD
      ;FOLD i4 ( F99 ) = i33 ;%{SE}%MKUKATPVW %CVW_SPS %VARIASG %P 2:i4 ( F99 ) = i33, 3: ARIASG
         VW(#COUNTER,$FLAG[99],4,$COUNT_I[33])
      ;ENDFOLD
      ;FOLD i1 ( EIN ) = 0 ;%{SE}%MKUKATPVW %CVW_SPS %VARIASG %P 2:i1 ( EIN ) = 0, 3: ARIASG
         VW(#COUNTER,TRUE,1,0)
      ;ENDFOLD
      ;FOLD F98 = AUS ;%{SE}%MKUKATPVW %CVW_SPS %VBOASG %P 2:F98 = AUS, 3: BOASG
         $FLAG[98] = FALSE
      ;ENDFOLD
      ;FOLD F312 = AUS ;%{SE}%MKUKATPVW %CVW_SPS %VBOASG %P 2:F312 = AUS, 3: BOASG
         $FLAG[312] = FALSE
      ;ENDFOLD
      ;FOLD F313 = AUS ;%{SE}%MKUKATPVW %CVW_SPS %VBOASG %P 2:F313 = AUS, 3: BOASG
         $FLAG[313] = FALSE
      ;ENDFOLD
      ;FOLD F324 = AUS ;%{SE}%MKUKATPVW %CVW_SPS %VBOASG %P 2:F324 = AUS, 3: BOASG
         $FLAG[324] = FALSE
      ;ENDFOLD
      ;FOLD F328 = AUS ;%{SE}%MKUKATPVW %CVW_SPS %VBOASG %P 2:F328 = AUS, 3: BOASG
         $FLAG[328] = FALSE
      ;ENDFOLD
      ;FOLD -- ServoGun Dress in Positon AUS -- ;%{SE}%MKUKATPVW %CVW_COM %VCOMMENT %P 2:-- ServoGun Dress in Positon AUS --, 3: VW_COMMENT
      ;ENDFOLD
      ;FOLD A3871 = AUS ;%{SE}%MKUKATPVW %CVW_SPS %VBOASG %P 2:A3871 = AUS, 3: BOASG
         $OUT[3871] = FALSE
      ;ENDFOLD
      ;FOLD -- KF1 einschalten nach Fehler -- ;%{SE}%MKUKATPVW %CVW_COM %VCOMMENT %P 2:-- KF1 einschalten nach Fehler --, 3: VW_COMMENT
      ;ENDFOLD
      ;FOLD A834 = EIN ;%{SE}%MKUKATPVW %CVW_SPS %VBOASG %P 2:A834 = EIN, 3: BOASG
         $OUT[834] = TRUE
      ;ENDFOLD
      ;FOLD -- KF1 Versetzeinheit rueck -- ;%{SE}%MKUKATPVW %CVW_COM %VCOMMENT %P 2:-- KF1 Versetzeinheit rueck --, 3: VW_COMMENT
      ;ENDFOLD
      ;FOLD A835 = AUS ;%{SE}%MKUKATPVW %CVW_SPS %VBOASG %P 2:A835 = AUS, 3: BOASG
         $OUT[835] = FALSE
      ;ENDFOLD
      ;FOLD bin30 ( EIN ) = p111 ;%{SE}%MKUKATPVW %CVW_SPS %VARIASG %P 2:bin30 ( EIN ) = p111, 3: ARIASG
         VW(#BINOUT,TRUE,30,PROCPAR[111])
      ;ENDFOLD
      ;FOLD -- Warte bis Fraeser in Position -- ;%{SE}%MKUKATPVW %CVW_COM %VCOMMENT %P 2:-- Warte bis Fraeser in Position --, 3: VW_COMMENT
      ;ENDFOLD
      ;FOLD Schritt 113 = T11 & !E836 & E837 & E838 & !E839 & A4039 ;%{SE}%MKUKATPVW %CVW_SPS %VST_CON %P 2:Schritt 113 = T11 & !E836 & E837 & E838 & !E839 & A4039, 3: ST_CON
         IF $TIMER_FLAG[11] AND NOT $IN[836] AND $IN[837] AND $IN[838] AND NOT $IN[839] AND $OUT[4039] THEN
            PREV_STEP[9] = APP_INT_STEP[9]
            APP_INT_STEP[9] = 113
         ENDIF
      ;ENDFOLD
      ;FOLD Schritt 113 = !E835 & !E836 & E837 & E838 & !E839 & A4039 ;%{SE}%MKUKATPVW %CVW_SPS %VST_CON %P 2:Schritt 113 = !E835 & !E836 & E837 & E838 & !E839 & A4039, 3: ST_CON
         IF NOT $IN[835] AND NOT $IN[836] AND $IN[837] AND $IN[838] AND NOT $IN[839] AND $OUT[4039] THEN
            PREV_STEP[9] = APP_INT_STEP[9]
            APP_INT_STEP[9] = 113
         ENDIF
      ;ENDFOLD
   ;ENDFOLD
   ;FOLD SCHRITT 113 -- st. RZ1 # DressInPos -- ;%{P}%MKUKATPVW,%CSTEP,%VST_NR,%P 1:SCHRITT, 2:113, 3: st. RZ1 # DressInPos
      ;FOLD ;%{H}
         Case 113
      ;ENDFOLD
      ;FOLD A840 = AUS ;%{SE}%MKUKATPVW %CVW_SPS %VBOASG %P 2:A840 = AUS, 3: BOASG
         $OUT[840] = FALSE
      ;ENDFOLD
      ;FOLD -- Ueberwachungszeit ServoGun SZ1 schliessen -- ;%{SE}%MKUKATPVW %CVW_COM %VCOMMENT %P 2:-- Ueberwachungszeit ServoGun SZ1 schliessen --, 3: VW_COMMENT
      ;ENDFOLD
      ;FOLD t9 ( EIN ) = -80[1/10Sek] ;%{SE}%MKUKATPVW %CVW_SPS %VTASG %P 2:t9 ( EIN ) = -80[1/10Sek], 3: TASG
         VW(#SET_TIME,TRUE,9,0,-80)
      ;ENDFOLD
      ;FOLD -- Verweilzeit Versetzeinheit Rueck -- ;%{SE}%MKUKATPVW %CVW_COM %VCOMMENT %P 2:-- Verweilzeit Versetzeinheit Rueck --, 3: VW_COMMENT
      ;ENDFOLD
      ;FOLD t11 ( EIN ) = STOP ;%{SE}%MKUKATPVW %CVW_SPS %VTSTOP %P 2:t11 ( EIN ) = STOP, 3: TSTOP
         VW(#SET_TIME,TRUE,11,1,0)
      ;ENDFOLD
      ;FOLD -- ServoGun SZ1 schliessen -- ;%{SE}%MKUKATPVW %CVW_COM %VCOMMENT %P 2:-- ServoGun SZ1 schliessen --, 3: VW_COMMENT
      ;ENDFOLD
      ;FOLD A3871 = !E836 & E837 & E838 & !E839 ;%{SE}%MKUKATPVW %CVW_SPS %VBOASG %P 2:A3871 = !E836 & E837 & E838 & !E839, 3: BOASG
         $OUT[3871] = NOT $IN[836] AND $IN[837] AND $IN[838] AND NOT $IN[839]
      ;ENDFOLD
      ;FOLD -- KF1 Ausblasen -- ;%{SE}%MKUKATPVW %CVW_COM %VCOMMENT %P 2:-- KF1 Ausblasen --, 3: VW_COMMENT
      ;ENDFOLD
      ;FOLD A836 = F330 + F331 + !F330 & !F331 & !F332 ;%{SE}%MKUKATPVW %CVW_SPS %VBOASG %P 2:A836 = F330 + F331 + !F330 & !F331 & !F332, 3: BOASG
         $OUT[836] = $FLAG[330] OR $FLAG[331] OR NOT $FLAG[330] AND NOT $FLAG[331] AND NOT $FLAG[332]
      ;ENDFOLD
      ;FOLD SCHRITT 114 = !A3862 & A3864 & A4039 + T9 ;%{SE}%MKUKATPVW %CVW_SPS %VST_CON %P 2:SCHRITT 114 = !A3862 & A3864 & A4039 + T9, 3: ST_CON
         IF NOT $OUT[3862] AND $OUT[3864] AND $OUT[4039] OR $TIMER_FLAG[9] THEN
            PREV_STEP[9] = APP_INT_STEP[9]
            APP_INT_STEP[9] = 114
         ENDIF
      ;ENDFOLD
      ;FOLD Schritt 150 = A3862 & !A3864 & A4039 & A3509 ;%{SE}%MKUKATPVW %CVW_SPS %VST_CON %P 2:Schritt 150 = A3862 & !A3864 & A4039 & A3509, 3: ST_CON
         IF $OUT[3862] AND NOT $OUT[3864] AND $OUT[4039] AND $OUT[3509] THEN
            PREV_STEP[9] = APP_INT_STEP[9]
            APP_INT_STEP[9] = 150
         ENDIF
      ;ENDFOLD
   ;ENDFOLD
   ;FOLD SCHRITT 114 -- st. RZ1 -- ;%{P}%MKUKATPVW,%CSTEP,%VST_NR,%P 1:SCHRITT, 2:114, 3: st. RZ1
      ;FOLD ;%{H}
         Case 114
      ;ENDFOLD
      ;FOLD -- RSK Fehlerausgabe Kraftaufbau -- ;%{SE}%MKUKATPVW %CVW_COM %VCOMMENT %P 2:-- RSK Fehlerausgabe Kraftaufbau --, 3: VW_COMMENT
      ;ENDFOLD
      ;FOLD F325 = T9 ;%{SE}%MKUKATPVW %CVW_SPS %VBOASG %P 2:F325 = T9, 3: BOASG
         $FLAG[325] = $TIMER_FLAG[9]
      ;ENDFOLD
      ;FOLD -- RSK Sammelstoerung -- ;%{SE}%MKUKATPVW %CVW_COM %VCOMMENT %P 2:-- RSK Sammelstoerung --, 3: VW_COMMENT
      ;ENDFOLD
      ;FOLD F329 = F325 ;%{SE}%MKUKATPVW %CVW_SPS %VBOASG %P 2:F329 = F325, 3: BOASG
         $FLAG[329] = $FLAG[325]
      ;ENDFOLD
      ;FOLD -- KF1 abschalten bei Fehler -- ;%{SE}%MKUKATPVW %CVW_COM %VCOMMENT %P 2:-- KF1 abschalten bei Fehler --, 3: VW_COMMENT
      ;ENDFOLD
      ;FOLD A834 = !T9 ;%{SE}%MKUKATPVW %CVW_SPS %VBOASG %P 2:A834 = !T9, 3: BOASG
         $OUT[834] = NOT $TIMER_FLAG[9]
      ;ENDFOLD
      ;FOLD -- KF1 Ausblasen -- ;%{SE}%MKUKATPVW %CVW_COM %VCOMMENT %P 2:-- KF1 Ausblasen --, 3: VW_COMMENT
      ;ENDFOLD
      ;FOLD A836 = (F330 + F331 + !F330 & !F331 & !F332) & !T9 ;%{SE}%MKUKATPVW %CVW_SPS %VBOASG %P 2:A836 = (F330 + F331 + !F330 & !F331 & !F332) & !T9, 3: BOASG
         $OUT[836] = ($FLAG[330] OR $FLAG[331] OR NOT $FLAG[330] AND NOT $FLAG[331] AND NOT $FLAG[332]) AND NOT $TIMER_FLAG[9]
      ;ENDFOLD
      ;FOLD -- Ueberwachungszeit Fehler Fraesen -- ;%{SE}%MKUKATPVW %CVW_COM %VCOMMENT %P 2:-- Ueberwachungszeit Fehler Fraesen --, 3: VW_COMMENT
      ;ENDFOLD
      ;FOLD t11 ( EIN ) = -110 [1/10Sek] ;%{SE}%MKUKATPVW %CVW_SPS %VTASG %P 2:t11 ( EIN ) = -110 [1/10Sek], 3: TASG
         VW(#SET_TIME,TRUE,11,0,-110)
      ;ENDFOLD
      ;FOLD -- Warte Fraesen fertig oder Timeout -- ;%{SE}%MKUKATPVW %CVW_COM %VCOMMENT %P 2:-- Warte Fraesen fertig oder Timeout --, 3: VW_COMMENT
      ;ENDFOLD
      ;FOLD SCHRITT 115 = (F79 & F98 + F78 & F94 & !F287 + T7 + T9 + F325) & A4039 ;%{SE}%MKUKATPVW %CVW_SPS %VST_CON %P 2:SCHRITT 115 = (F79 & F98 + F78 & F94 & !F287 + T7 + T9 + F325) & A4039, 3: ST_CON
         IF ($FLAG[79] AND $FLAG[98] OR $FLAG[78] AND $FLAG[94] AND NOT $FLAG[287] OR $TIMER_FLAG[7] OR $TIMER_FLAG[9] OR $FLAG[325]) AND $OUT[4039] THEN
            PREV_STEP[9] = APP_INT_STEP[9]
            APP_INT_STEP[9] = 115
         ENDIF
      ;ENDFOLD
      ;FOLD SCHRITT 115 = (F78 & F96 & F287 + T7 + T9 + F325) & A4039 ;%{SE}%MKUKATPVW %CVW_SPS %VST_CON %P 2:SCHRITT 115 = (F78 & F96 & F287 + T7 + T9 + F325) & A4039, 3: ST_CON
         IF ($FLAG[78] AND $FLAG[96] AND $FLAG[287] OR $TIMER_FLAG[7] OR $TIMER_FLAG[9] OR $FLAG[325]) AND $OUT[4039] THEN
            PREV_STEP[9] = APP_INT_STEP[9]
            APP_INT_STEP[9] = 115
         ENDIF
      ;ENDFOLD
   ;ENDFOLD
   ;FOLD SCHRITT 115 -- st. RZ1 # GunOpen -- ;%{P}%MKUKATPVW,%CSTEP,%VST_NR,%P 1:SCHRITT, 2:115, 3: st. RZ1 # GunOpen
      ;FOLD ;%{H}
         Case 115
      ;ENDFOLD
      ;FOLD -- ServoGun SZ1 oeffnen -- ;%{SE}%MKUKATPVW %CVW_COM %VCOMMENT %P 2:-- ServoGun SZ1 oeffnen --, 3: VW_COMMENT
      ;ENDFOLD
      ;FOLD t9 ( EIN ) = STOP ;%{SE}%MKUKATPVW %CVW_SPS %VTSTOP %P 2:t9 ( EIN ) = STOP, 3: TSTOP
         VW(#SET_TIME,TRUE,9,1,0)
      ;ENDFOLD
      ;FOLD A3871 = AUS ;%{SE}%MKUKATPVW %CVW_SPS %VBOASG %P 2:A3871 = AUS, 3: BOASG
         $OUT[3871] = FALSE
      ;ENDFOLD
      ;FOLD A3872 = EIN ;%{SE}%MKUKATPVW %CVW_SPS %VBOASG %P 2:A3872 = EIN, 3: BOASG
         $OUT[3872] = TRUE
      ;ENDFOLD
      ;FOLD -- KF1 Ausblasen -- ;%{SE}%MKUKATPVW %CVW_COM %VCOMMENT %P 2:-- KF1 Ausblasen --, 3: VW_COMMENT
      ;ENDFOLD
      ;FOLD A836 = (F330 + F331 + F332 + !F330 & !F331 & !F332) & !T9 ;%{SE}%MKUKATPVW %CVW_SPS %VBOASG %P 2:A836 = (F330 + F331 + F332 + !F330 & !F331 & !F332) & !T9, 3: BOASG
         $OUT[836] = ($FLAG[330] OR $FLAG[331] OR $FLAG[332] OR NOT $FLAG[330] AND NOT $FLAG[331] AND NOT $FLAG[332]) AND NOT $TIMER_FLAG[9]
      ;ENDFOLD
      ;FOLD -- KF Ausblasen Ausschaltverzoegerung starten -- ;%{SE}%MKUKATPVW %CVW_COM %VCOMMENT %P 2:-- KF Ausblasen Ausschaltverzoegerung starten --, 3: VW_COMMENT
      ;ENDFOLD
      ;FOLD F737 = AUS ;%{SE}%MKUKATPVW %CVW_SPS %VBOASG %P 2:F737 = AUS, 3: BOASG
         $FLAG[737] = FALSE
      ;ENDFOLD
      ;FOLD -- RSK Sammelstoerung -- ;%{SE}%MKUKATPVW %CVW_COM %VCOMMENT %P 2:-- RSK Sammelstoerung --, 3: VW_COMMENT
      ;ENDFOLD
      ;FOLD F329 = T7 + T9 + F325 ;%{SE}%MKUKATPVW %CVW_SPS %VBOASG %P 2:F329 = T7 + T9 + F325, 3: BOASG
         $FLAG[329] = $TIMER_FLAG[7] OR $TIMER_FLAG[9] OR $FLAG[325]
      ;ENDFOLD
      ;FOLD -- Hilfsflag Startfraesen -- ;%{SE}%MKUKATPVW %CVW_COM %VCOMMENT %P 2:-- Hilfsflag Startfraesen --, 3: VW_COMMENT
      ;ENDFOLD
      ;FOLD F96 = F96 & F287 ;%{SE}%MKUKATPVW %CVW_SPS %VBOASG %P 2:F96 = F96 & F287, 3: BOASG
         $FLAG[96] = $FLAG[96] AND $FLAG[287]
      ;ENDFOLD
      ;FOLD F96 = (F96 & F78 + F98 & F79) & F287 ;%{SE}%MKUKATPVW %CVW_SPS %VBOASG %P 2:F96 = (F96 & F78 + F98 & F79) & F287, 3: BOASG
         $FLAG[96] = ($FLAG[96] AND $FLAG[78] OR $FLAG[98] AND $FLAG[79]) AND $FLAG[287]
      ;ENDFOLD
      ;FOLD F98 = !F130 & F98 + F130 & F287 & F98 ;%{SE}%MKUKATPVW %CVW_SPS %VBOASG %P 2:F98 = !F130 & F98 + F130 & F287 & F98, 3: BOASG
         $FLAG[98] = NOT $FLAG[130] AND $FLAG[98] OR $FLAG[130] AND $FLAG[287] AND $FLAG[98]
      ;ENDFOLD
      ;FOLD F287 = F78 + F79 & F130 ;%{SE}%MKUKATPVW %CVW_SPS %VBOASG %P 2:F287 = F78 + F79 & F130, 3: BOASG
         $FLAG[287] = $FLAG[78] OR $FLAG[79] AND $FLAG[130]
      ;ENDFOLD
      ;FOLD -- Neues Fraesprogramm und Zaehler ruecksetzen -- ;%{SE}%MKUKATPVW %CVW_COM %VCOMMENT %P 2:-- Neues Fraesprogramm und Zaehler ruecksetzen --, 3: VW_COMMENT
      ;ENDFOLD
      ;FOLD bin31 ( F130 ) = 36 ;%{SE}%MKUKATPVW %CVW_SPS %VARIASG %P 2:bin31 ( F130 ) = 36, 3: ARIASG
         VW(#BINOUT,$FLAG[130],31,36)
      ;ENDFOLD
      ;FOLD i4 ( F96 ) = i45 ;%{SE}%MKUKATPVW %CVW_SPS %VARIASG %P 2:i4 ( F96 ) = i45, 3: ARIASG
         VW(#COUNTER,$FLAG[96],4,$COUNT_I[45])
      ;ENDFOLD
      ;FOLD -- Fehler Fraesen -- ;%{SE}%MKUKATPVW %CVW_COM %VCOMMENT %P 2:-- Fehler Fraesen --, 3: VW_COMMENT
      ;ENDFOLD
      ;FOLD Schritt 150 = (!A3862 & !A3508 & T11) + (A3862 & !A3508 & T11) & A4039 ;%{SE}%MKUKATPVW %CVW_SPS %VST_CON %P 2:Schritt 150 = (!A3862 & !A3508 & T11) + (A3862 & !A3508 & T11) & A4039, 3: ST_CON
         IF (NOT $OUT[3862] AND NOT $OUT[3508] AND $TIMER_FLAG[11]) OR ($OUT[3862] AND NOT $OUT[3508] AND $TIMER_FLAG[11]) AND $OUT[4039] THEN
            PREV_STEP[9] = APP_INT_STEP[9]
            APP_INT_STEP[9] = 150
         ENDIF
      ;ENDFOLD
      ;FOLD -- Wiederholung beim Normalfraesen -- ;%{SE}%MKUKATPVW %CVW_COM %VCOMMENT %P 2:-- Wiederholung beim Normalfraesen --, 3: VW_COMMENT
      ;ENDFOLD
      ;FOLD Schritt 111 = A3862 & A3508 & (!F78 & F79 & F130 & !F96) & !F329 & A4039 ;%{SE}%MKUKATPVW %CVW_SPS %VST_CON %P 2:Schritt 111 = A3862 & A3508 & (!F78 & F79 & F130 & !F96) & !F329 & A4039, 3: ST_CON
         IF $OUT[3862] AND $OUT[3508] AND (NOT $FLAG[78] AND $FLAG[79] AND $FLAG[130] AND NOT $FLAG[96]) AND NOT $FLAG[329] AND $OUT[4039] THEN
            PREV_STEP[9] = APP_INT_STEP[9]
            APP_INT_STEP[9] = 111
         ENDIF
      ;ENDFOLD
      ;FOLD -- Wiederholung beim Startfraesen -- ;%{SE}%MKUKATPVW %CVW_COM %VCOMMENT %P 2:-- Wiederholung beim Startfraesen --, 3: VW_COMMENT
      ;ENDFOLD
      ;FOLD Schritt 111 = A3862 & A3508 & (F78 & !F96 + F79 & F130 & !F96) & !F329 & A4039 & A3520 ;%{SE}%MKUKATPVW %CVW_SPS %VST_CON %P 2:Schritt 111 = A3862 & A3508 & (F78 & !F96 + F79 & F130 & !F96) & !F329 & A4039 & A3520, 3: ST_CON
         IF $OUT[3862] AND $OUT[3508] AND ($FLAG[78] AND NOT $FLAG[96] OR $FLAG[79] AND $FLAG[130] AND NOT $FLAG[96]) AND NOT $FLAG[329] AND $OUT[4039] AND $OUT[3520] THEN
            PREV_STEP[9] = APP_INT_STEP[9]
            APP_INT_STEP[9] = 111
         ENDIF
      ;ENDFOLD
      ;FOLD -- Wiederholung beim Startfraesen -- ;%{SE}%MKUKATPVW %CVW_COM %VCOMMENT %P 2:-- Wiederholung beim Startfraesen --, 3: VW_COMMENT
      ;ENDFOLD
      ;FOLD Schritt 116 = A3862 & A3508 & (F78 & !F96 + F79 & F130 & F96) & !F329 & A4039 & !A3520 ;%{SE}%MKUKATPVW %CVW_SPS %VST_CON %P 2:Schritt 116 = A3862 & A3508 & (F78 & !F96 + F79 & F130 & F96) & !F329 & A4039 & !A3520, 3: ST_CON
         IF $OUT[3862] AND $OUT[3508] AND ($FLAG[78] AND NOT $FLAG[96] OR $FLAG[79] AND $FLAG[130] AND $FLAG[96]) AND NOT $FLAG[329] AND $OUT[4039] AND NOT $OUT[3520] THEN
            PREV_STEP[9] = APP_INT_STEP[9]
            APP_INT_STEP[9] = 116
         ENDIF
      ;ENDFOLD
      ;FOLD -- Weiter wenn Fraesen fertig -- ;%{SE}%MKUKATPVW %CVW_COM %VCOMMENT %P 2:-- Weiter wenn Fraesen fertig --, 3: VW_COMMENT
      ;ENDFOLD
      ;FOLD Schritt 116 = A3862 & A3508 & (F79 & F98 & (!F130 + F96) + F78 & F96 + F329) & A4039 ;%{SE}%MKUKATPVW %CVW_SPS %VST_CON %P 2:Schritt 116 = A3862 & A3508 & (F79 & F98 & (!F130 + F96) + F78 & F96 + F329) & A4039, 3: ST_CON
         IF $OUT[3862] AND $OUT[3508] AND ($FLAG[79] AND $FLAG[98] AND (NOT $FLAG[130] OR $FLAG[96]) OR $FLAG[78] AND $FLAG[96] OR $FLAG[329]) AND $OUT[4039] THEN
            PREV_STEP[9] = APP_INT_STEP[9]
            APP_INT_STEP[9] = 116
         ENDIF
      ;ENDFOLD
   ;ENDFOLD
   ;FOLD SCHRITT 116 -- st. RZ1 # Acknowledge -- ;%{P}%MKUKATPVW,%CSTEP,%VST_NR,%P 1:SCHRITT, 2:116, 3: st. RZ1 # Acknowledge
      ;FOLD ;%{H}
         Case 116
      ;ENDFOLD
      ;FOLD -- Hilfsflag Durchlaufmerker -- ;%{SE}%MKUKATPVW %CVW_COM %VCOMMENT %P 2:-- Hilfsflag Durchlaufmerker --, 3: VW_COMMENT
      ;ENDFOLD
      ;FOLD F324 = AUS ;%{SE}%MKUKATPVW %CVW_SPS %VBOASG %P 2:F324 = AUS, 3: BOASG
         $FLAG[324] = FALSE
      ;ENDFOLD
      ;FOLD A3871 = AUS ;%{SE}%MKUKATPVW %CVW_SPS %VBOASG %P 2:A3871 = AUS, 3: BOASG
         $OUT[3871] = FALSE
      ;ENDFOLD
      ;FOLD A3872 = AUS ;%{SE}%MKUKATPVW %CVW_SPS %VBOASG %P 2:A3872 = AUS, 3: BOASG
         $OUT[3872] = FALSE
      ;ENDFOLD
      ;FOLD A3510 = AUS ;%{SE}%MKUKATPVW %CVW_SPS %VBOASG %P 2:A3510 = AUS, 3: BOASG
         $OUT[3510] = FALSE
      ;ENDFOLD
      ;FOLD A3512 = EIN ;%{SE}%MKUKATPVW %CVW_SPS %VBOASG %P 2:A3512 = EIN, 3: BOASG
         $OUT[3512] = TRUE
      ;ENDFOLD
      ;FOLD t9 ( EIN ) = STOP ;%{SE}%MKUKATPVW %CVW_SPS %VTSTOP %P 2:t9 ( EIN ) = STOP, 3: TSTOP
         VW(#SET_TIME,TRUE,9,1,0)
      ;ENDFOLD
      ;FOLD -- KF1 abschalten -- ;%{SE}%MKUKATPVW %CVW_COM %VCOMMENT %P 2:-- KF1 abschalten --, 3: VW_COMMENT
      ;ENDFOLD
      ;FOLD A834 = AUS ;%{SE}%MKUKATPVW %CVW_SPS %VBOASG %P 2:A834 = AUS, 3: BOASG
         $OUT[834] = FALSE
      ;ENDFOLD
      ;FOLD -- Ueberwachungszeit KF1 Versetzeinheit -- ;%{SE}%MKUKATPVW %CVW_COM %VCOMMENT %P 2:-- Ueberwachungszeit KF1 Versetzeinheit --, 3: VW_COMMENT
      ;ENDFOLD
      ;FOLD t8 ( EIN ) = -40[1/10Sek] ;%{SE}%MKUKATPVW %CVW_SPS %VTASG %P 2:t8 ( EIN ) = -40[1/10Sek], 3: TASG
         VW(#SET_TIME,TRUE,8,0,-40)
      ;ENDFOLD
      ;FOLD SCHRITT 117 = A4039 & !E195 ;%{SE}%MKUKATPVW %CVW_SPS %VST_CON %P 2:SCHRITT 117 = A4039 & !E195, 3: ST_CON
         IF $OUT[4039] AND NOT $IN[195] THEN
            PREV_STEP[9] = APP_INT_STEP[9]
            APP_INT_STEP[9] = 117
         ENDIF
      ;ENDFOLD
   ;ENDFOLD
   ;FOLD SCHRITT 117 -- st. RZ1 -- ;%{P}%MKUKATPVW,%CSTEP,%VST_NR,%P 1:SCHRITT, 2:117, 3: st. RZ1
      ;FOLD ;%{H}
         Case 117
      ;ENDFOLD
      ;FOLD -- RSK Fehlerausgabe Arbeitsst. -- ;%{SE}%MKUKATPVW %CVW_COM %VCOMMENT %P 2:-- RSK Fehlerausgabe Arbeitsst. --, 3: VW_COMMENT
      ;ENDFOLD
      ;FOLD F328 = AUS ;%{SE}%MKUKATPVW %CVW_SPS %VBOASG %P 2:F328 = AUS, 3: BOASG
         $FLAG[328] = FALSE
      ;ENDFOLD
      ;FOLD -- KF1 Versetzeinheit vor -- ;%{SE}%MKUKATPVW %CVW_COM %VCOMMENT %P 2:-- KF1 Versetzeinheit vor --, 3: VW_COMMENT
      ;ENDFOLD
      ;FOLD A835 = F564 ;%{SE}%MKUKATPVW %CVW_SPS %VBOASG %P 2:A835 = F564, 3: BOASG
         $OUT[835] = $FLAG[564]
      ;ENDFOLD
      ;FOLD A3512 = AUS ;%{SE}%MKUKATPVW %CVW_SPS %VBOASG %P 2:A3512 = AUS, 3: BOASG
         $OUT[3512] = FALSE
      ;ENDFOLD
      ;FOLD -- RSK Fehlerausgabe KS1 Arbeitsst. -- ;%{SE}%MKUKATPVW %CVW_COM %VCOMMENT %P 2:-- RSK Fehlerausgabe KS1 Arbeitsst. --, 3: VW_COMMENT
      ;ENDFOLD
      ;FOLD F324 = (E836 + !E837 + !E838 + E839) & !F323 & !F328 + F324 ;%{SE}%MKUKATPVW %CVW_SPS %VBOASG %P 2:F324 = (E836 + !E837 + !E838 + E839) & !F323 & !F328 + F324, 3: BOASG
         $FLAG[324] = ($IN[836] OR NOT $IN[837] OR NOT $IN[838] OR $IN[839]) AND NOT $FLAG[323] AND NOT $FLAG[328] OR $FLAG[324]
      ;ENDFOLD
      ;FOLD -- RSK Sammelstoerung -- ;%{SE}%MKUKATPVW %CVW_COM %VCOMMENT %P 2:-- RSK Sammelstoerung --, 3: VW_COMMENT
      ;ENDFOLD
      ;FOLD F329 = F324 + F325 ;%{SE}%MKUKATPVW %CVW_SPS %VBOASG %P 2:F329 = F324 + F325, 3: BOASG
         $FLAG[329] = $FLAG[324] OR $FLAG[325]
      ;ENDFOLD
      ;FOLD -- Ueberwachungszeit KS1 schwenken -- ;%{SE}%MKUKATPVW %CVW_COM %VCOMMENT %P 2:-- Ueberwachungszeit KS1 schwenken --, 3: VW_COMMENT
      ;ENDFOLD
      ;FOLD t9 ( EIN ) = -100[1/10Sek] ;%{SE}%MKUKATPVW %CVW_SPS %VTASG %P 2:t9 ( EIN ) = -100[1/10Sek], 3: TASG
         VW(#SET_TIME,TRUE,9,0,-100)
      ;ENDFOLD
      ;FOLD SCHRITT 116 = F324 & (E26 + E27) & A4039 ;%{SE}%MKUKATPVW %CVW_SPS %VST_CON %P 2:SCHRITT 116 = F324 & (E26 + E27) & A4039, 3: ST_CON
         IF $FLAG[324] AND ($IN[26] OR $IN[27]) AND $OUT[4039] THEN
            PREV_STEP[9] = APP_INT_STEP[9]
            APP_INT_STEP[9] = 116
         ENDIF
      ;ENDFOLD
      ;FOLD SCHRITT 118 = (!F324 & (E835 & F564 + !E835 & !F564) + T8 + F325) & A4039 ;%{SE}%MKUKATPVW %CVW_SPS %VST_CON %P 2:SCHRITT 118 = (!F324 & (E835 & F564 + !E835 & !F564) + T8 + F325) & A4039, 3: ST_CON
         IF (NOT $FLAG[324] AND ($IN[835] AND $FLAG[564] OR NOT $IN[835] AND NOT $FLAG[564]) OR $TIMER_FLAG[8] OR $FLAG[325]) AND $OUT[4039] THEN
            PREV_STEP[9] = APP_INT_STEP[9]
            APP_INT_STEP[9] = 118
         ENDIF
      ;ENDFOLD
   ;ENDFOLD
   ;FOLD SCHRITT 118 -- st. RZ1 # KS in RS schwenken -- ;%{P}%MKUKATPVW,%CSTEP,%VST_NR,%P 1:SCHRITT, 2:118, 3: st. RZ1 # KS in RS schwenken
      ;FOLD ;%{H}
         Case 118
      ;ENDFOLD
      ;FOLD F323 = AUS ;%{SE}%MKUKATPVW %CVW_SPS %VBOASG %P 2:F323 = AUS, 3: BOASG
         $FLAG[323] = FALSE
      ;ENDFOLD
      ;FOLD F328 = AUS ;%{SE}%MKUKATPVW %CVW_SPS %VBOASG %P 2:F328 = AUS, 3: BOASG
         $FLAG[328] = FALSE
      ;ENDFOLD
      ;FOLD -- RSK Sammelstoerung -- ;%{SE}%MKUKATPVW %CVW_COM %VCOMMENT %P 2:-- RSK Sammelstoerung --, 3: VW_COMMENT
      ;ENDFOLD
      ;FOLD F329 = F325 ;%{SE}%MKUKATPVW %CVW_SPS %VBOASG %P 2:F329 = F325, 3: BOASG
         $FLAG[329] = $FLAG[325]
      ;ENDFOLD
      ;FOLD -- KF1 ein -- ;%{SE}%MKUKATPVW %CVW_COM %VCOMMENT %P 2:-- KF1 ein --, 3: VW_COMMENT
      ;ENDFOLD
      ;FOLD A834 = EIN ;%{SE}%MKUKATPVW %CVW_SPS %VBOASG %P 2:A834 = EIN, 3: BOASG
         $OUT[834] = TRUE
      ;ENDFOLD
      ;FOLD -- KF Ausblasen Ausschaltverzoegerung starten -- ;%{SE}%MKUKATPVW %CVW_COM %VCOMMENT %P 2:-- KF Ausblasen Ausschaltverzoegerung starten --, 3: VW_COMMENT
      ;ENDFOLD
      ;FOLD F737 = EIN ;%{SE}%MKUKATPVW %CVW_SPS %VBOASG %P 2:F737 = EIN, 3: BOASG
         $FLAG[737] = TRUE
      ;ENDFOLD
      ;FOLD -- KF1 Ausblasen -- ;%{SE}%MKUKATPVW %CVW_COM %VCOMMENT %P 2:-- KF1 Ausblasen --, 3: VW_COMMENT
      ;ENDFOLD
      ;FOLD A836 = (F330 + F331 + F332) & F737 ;%{SE}%MKUKATPVW %CVW_SPS %VBOASG %P 2:A836 = (F330 + F331 + F332) & F737, 3: BOASG
         $OUT[836] = ($FLAG[330] OR $FLAG[331] OR $FLAG[332]) AND $FLAG[737]
      ;ENDFOLD
      ;FOLD -- KS1 in Ruhestellung schwenken -- ;%{SE}%MKUKATPVW %CVW_COM %VCOMMENT %P 2:-- KS1 in Ruhestellung schwenken --, 3: VW_COMMENT
      ;ENDFOLD
      ;FOLD A840 = A3862 & (E835 & F564 + !E835 & !F564) ;%{SE}%MKUKATPVW %CVW_SPS %VBOASG %P 2:A840 = A3862 & (E835 & F564 + !E835 & !F564), 3: BOASG
         $OUT[840] = $OUT[3862] AND ($IN[835] AND $FLAG[564] OR NOT $IN[835] AND NOT $FLAG[564])
      ;ENDFOLD
      ;FOLD Schritt 120 = A3862 & A840 & A4039 + T9 ;%{SE}%MKUKATPVW %CVW_SPS %VST_CON %P 2:Schritt 120 = A3862 & A840 & A4039 + T9, 3: ST_CON
         IF $OUT[3862] AND $OUT[840] AND $OUT[4039] OR $TIMER_FLAG[9] THEN
            PREV_STEP[9] = APP_INT_STEP[9]
            APP_INT_STEP[9] = 120
         ENDIF
      ;ENDFOLD
   ;ENDFOLD
   ;FOLD SCHRITT 120 -- st. RZ1 -- ;%{P}%MKUKATPVW,%CSTEP,%VST_NR,%P 1:SCHRITT, 2:120, 3: st. RZ1
      ;FOLD ;%{H}
         Case 120
      ;ENDFOLD
      ;FOLD -- Hilfsflag SK Programmwechsel -- ;%{SE}%MKUKATPVW %CVW_COM %VCOMMENT %P 2:-- Hilfsflag SK Programmwechsel --, 3: VW_COMMENT
      ;ENDFOLD
      ;FOLD F334 = AUS ;%{SE}%MKUKATPVW %CVW_SPS %VBOASG %P 2:F334 = AUS, 3: BOASG
         $FLAG[334] = FALSE
      ;ENDFOLD
      ;FOLD -- RSK Fehlerausgabe KF Versetzeinheit -- ;%{SE}%MKUKATPVW %CVW_COM %VCOMMENT %P 2:-- RSK Fehlerausgabe KF Versetzeinheit --, 3: VW_COMMENT
      ;ENDFOLD
      ;FOLD F328 = !E835 & F564 & !F323 + F328 ;%{SE}%MKUKATPVW %CVW_SPS %VBOASG %P 2:F328 = !E835 & F564 & !F323 + F328, 3: BOASG
         $FLAG[328] = NOT $IN[835] AND $FLAG[564] AND NOT $FLAG[323] OR $FLAG[328]
      ;ENDFOLD
      ;FOLD -- RSK Fehlerausgabe KS1 Ruhestellung -- ;%{SE}%MKUKATPVW %CVW_COM %VCOMMENT %P 2:-- RSK Fehlerausgabe KS1 Ruhestellung --, 3: VW_COMMENT
      ;ENDFOLD
      ;FOLD F323 = (!E836 + E837 + E838 + !E839) & T9 & (E835 + !F564) + F323 ;%{SE}%MKUKATPVW %CVW_SPS %VBOASG %P 2:F323 = (!E836 + E837 + E838 + !E839) & T9 & (E835 + !F564) + F323, 3: BOASG
         $FLAG[323] = (NOT $IN[836] OR $IN[837] OR $IN[838] OR NOT $IN[839]) AND $TIMER_FLAG[9] AND ($IN[835] OR NOT $FLAG[564]) OR $FLAG[323]
      ;ENDFOLD
      ;FOLD -- RSK Fehlerausgabe EZ/SP min. Oeffnung -- ;%{SE}%MKUKATPVW %CVW_COM %VCOMMENT %P 2:-- RSK Fehlerausgabe EZ/SP min. Oeffnung --, 3: VW_COMMENT
      ;ENDFOLD
      ;FOLD F333 = !A3862 ;%{SE}%MKUKATPVW %CVW_SPS %VBOASG %P 2:F333 = !A3862, 3: BOASG
         $FLAG[333] = NOT $OUT[3862]
      ;ENDFOLD
      ;FOLD -- RSK Sammelstoerung -- ;%{SE}%MKUKATPVW %CVW_COM %VCOMMENT %P 2:-- RSK Sammelstoerung --, 3: VW_COMMENT
      ;ENDFOLD
      ;FOLD F329 = F323 + F325 + F328 + F333 ;%{SE}%MKUKATPVW %CVW_SPS %VBOASG %P 2:F329 = F323 + F325 + F328 + F333, 3: BOASG
         $FLAG[329] = $FLAG[323] OR $FLAG[325] OR $FLAG[328] OR $FLAG[333]
      ;ENDFOLD
      ;FOLD A834 = !F329 ;%{SE}%MKUKATPVW %CVW_SPS %VBOASG %P 2:A834 = !F329, 3: BOASG
         $OUT[834] = NOT $FLAG[329]
      ;ENDFOLD
      ;FOLD A835 = F564 ;%{SE}%MKUKATPVW %CVW_SPS %VBOASG %P 2:A835 = F564, 3: BOASG
         $OUT[835] = $FLAG[564]
      ;ENDFOLD
      ;FOLD SCHRITT 116 = (F323 + F328) & (E26 + E27) & A4039 ;%{SE}%MKUKATPVW %CVW_SPS %VST_CON %P 2:SCHRITT 116 = (F323 + F328) & (E26 + E27) & A4039, 3: ST_CON
         IF ($FLAG[323] OR $FLAG[328]) AND ($IN[26] OR $IN[27]) AND $OUT[4039] THEN
            PREV_STEP[9] = APP_INT_STEP[9]
            APP_INT_STEP[9] = 116
         ENDIF
      ;ENDFOLD
      ;FOLD Schritt 121 = (!A840 + A840) & E836 & !E837 & !E838 & E839 & A4039 ;%{SE}%MKUKATPVW %CVW_SPS %VST_CON %P 2:Schritt 121 = (!A840 + A840) & E836 & !E837 & !E838 & E839 & A4039, 3: ST_CON
         IF (NOT $OUT[840] OR $OUT[840]) AND $IN[836] AND NOT $IN[837] AND NOT $IN[838] AND $IN[839] AND $OUT[4039] THEN
            PREV_STEP[9] = APP_INT_STEP[9]
            APP_INT_STEP[9] = 121
         ENDIF
      ;ENDFOLD
   ;ENDFOLD
   ;FOLD SCHRITT 121 -- st. RZ1 -- ;%{P}%MKUKATPVW,%CSTEP,%VST_NR,%P 1:SCHRITT, 2:121, 3: st. RZ1
      ;FOLD ;%{H}
         Case 121
      ;ENDFOLD
      ;FOLD A840 = AUS ;%{SE}%MKUKATPVW %CVW_SPS %VBOASG %P 2:A840 = AUS, 3: BOASG
         $OUT[840] = FALSE
      ;ENDFOLD
      ;FOLD F323 = AUS ;%{SE}%MKUKATPVW %CVW_SPS %VBOASG %P 2:F323 = AUS, 3: BOASG
         $FLAG[323] = FALSE
      ;ENDFOLD
      ;FOLD F328 = AUS ;%{SE}%MKUKATPVW %CVW_SPS %VBOASG %P 2:F328 = AUS, 3: BOASG
         $FLAG[328] = FALSE
      ;ENDFOLD
      ;FOLD -- KF Ausblasen Ausschaltverzoegerung starten -- ;%{SE}%MKUKATPVW %CVW_COM %VCOMMENT %P 2:-- KF Ausblasen Ausschaltverzoegerung starten --, 3: VW_COMMENT
      ;ENDFOLD
      ;FOLD F737 = EIN ;%{SE}%MKUKATPVW %CVW_SPS %VBOASG %P 2:F737 = EIN, 3: BOASG
         $FLAG[737] = TRUE
      ;ENDFOLD
      ;FOLD -- RSK Sammelstoerung -- ;%{SE}%MKUKATPVW %CVW_COM %VCOMMENT %P 2:-- RSK Sammelstoerung --, 3: VW_COMMENT
      ;ENDFOLD
      ;FOLD F329 = F325 ;%{SE}%MKUKATPVW %CVW_SPS %VBOASG %P 2:F329 = F325, 3: BOASG
         $FLAG[329] = $FLAG[325]
      ;ENDFOLD
      ;FOLD t9 ( EIN ) = STOP ;%{SE}%MKUKATPVW %CVW_SPS %VTSTOP %P 2:t9 ( EIN ) = STOP, 3: TSTOP
         VW(#SET_TIME,TRUE,9,1,0)
      ;ENDFOLD
      ;FOLD -- KF1 Versetzeinheit rueck -- ;%{SE}%MKUKATPVW %CVW_COM %VCOMMENT %P 2:-- KF1 Versetzeinheit rueck --, 3: VW_COMMENT
      ;ENDFOLD
      ;FOLD A835 = AUS ;%{SE}%MKUKATPVW %CVW_SPS %VBOASG %P 2:A835 = AUS, 3: BOASG
         $OUT[835] = FALSE
      ;ENDFOLD
      ;FOLD -- KF1 aus -- ;%{SE}%MKUKATPVW %CVW_COM %VCOMMENT %P 2:-- KF1 aus --, 3: VW_COMMENT
      ;ENDFOLD
      ;FOLD A834 = AUS ;%{SE}%MKUKATPVW %CVW_SPS %VBOASG %P 2:A834 = AUS, 3: BOASG
         $OUT[834] = FALSE
      ;ENDFOLD
      ;FOLD -- KF1 Ausblasen AUS -- ;%{SE}%MKUKATPVW %CVW_COM %VCOMMENT %P 2:-- KF1 Ausblasen AUS --, 3: VW_COMMENT
      ;ENDFOLD
      ;FOLD A836 = AUS ;%{SE}%MKUKATPVW %CVW_SPS %VBOASG %P 2:A836 = AUS, 3: BOASG
         $OUT[836] = FALSE
      ;ENDFOLD
      ;FOLD bin1 ( !F329 ) = 1 ;%{SE}%MKUKATPVW %CVW_SPS %VARIASG %P 2:bin1 ( !F329 ) = 1, 3: ARIASG
         VW(#BINOUT,NOT $FLAG[329],1,1)
      ;ENDFOLD
      ;FOLD bin3 ( !F329 ) = 1 ;%{SE}%MKUKATPVW %CVW_SPS %VARIASG %P 2:bin3 ( !F329 ) = 1, 3: ARIASG
         VW(#BINOUT,NOT $FLAG[329],3,1)
      ;ENDFOLD
      ;FOLD bin31 ( !F329 ) = 1 ;%{SE}%MKUKATPVW %CVW_SPS %VARIASG %P 2:bin31 ( !F329 ) = 1, 3: ARIASG
         VW(#BINOUT,NOT $FLAG[329],31,1)
      ;ENDFOLD
      ;FOLD -- Wartezeit Programmwechsel SK -- ;%{SE}%MKUKATPVW %CVW_COM %VCOMMENT %P 2:-- Wartezeit Programmwechsel SK --, 3: VW_COMMENT
      ;ENDFOLD
      ;FOLD T8 ( !F334 ) = -2[1/10Sek] ;%{SE}%MKUKATPVW %CVW_SPS %VTASG %P 2:T8 ( !F334 ) = -2[1/10Sek], 3: TASG
         VW(#SET_TIME,NOT $FLAG[334],8,0,-2)
      ;ENDFOLD
      ;FOLD -- Hilfsflag SK Programmwechsel -- ;%{SE}%MKUKATPVW %CVW_COM %VCOMMENT %P 2:-- Hilfsflag SK Programmwechsel --, 3: VW_COMMENT
      ;ENDFOLD
      ;FOLD F334 = EIN ;%{SE}%MKUKATPVW %CVW_SPS %VBOASG %P 2:F334 = EIN, 3: BOASG
         $FLAG[334] = TRUE
      ;ENDFOLD
      ;FOLD Schritt 103 = (F325 + F329) & (E26 + E27) & A4039 ;%{SE}%MKUKATPVW %CVW_SPS %VST_CON %P 2:Schritt 103 = (F325 + F329) & (E26 + E27) & A4039, 3: ST_CON
         IF ($FLAG[325] OR $FLAG[329]) AND ($IN[26] OR $IN[27]) AND $OUT[4039] THEN
            PREV_STEP[9] = APP_INT_STEP[9]
            APP_INT_STEP[9] = 103
         ENDIF
      ;ENDFOLD
      ;FOLD SCHRITT 122 = T8 & !F325 & !F329 & A4039 & (A3506 & A3505) ;%{SE}%MKUKATPVW %CVW_SPS %VST_CON %P 2:SCHRITT 122 = T8 & !F325 & !F329 & A4039 & (A3506 & A3505), 3: ST_CON
         IF $TIMER_FLAG[8] AND NOT $FLAG[325] AND NOT $FLAG[329] AND $OUT[4039] AND ($OUT[3506] AND $OUT[3505]) THEN
            PREV_STEP[9] = APP_INT_STEP[9]
            APP_INT_STEP[9] = 122
         ENDIF
      ;ENDFOLD
   ;ENDFOLD
   ;FOLD SCHRITT 122 -- st. RZ1 -- ;%{P}%MKUKATPVW,%CSTEP,%VST_NR,%P 1:SCHRITT, 2:122, 3: st. RZ1
      ;FOLD ;%{H}
         Case 122
      ;ENDFOLD
      ;FOLD -- Hilfsflag SK Programmwechsel -- ;%{SE}%MKUKATPVW %CVW_COM %VCOMMENT %P 2:-- Hilfsflag SK Programmwechsel --, 3: VW_COMMENT
      ;ENDFOLD
      ;FOLD F334 = AUS ;%{SE}%MKUKATPVW %CVW_SPS %VBOASG %P 2:F334 = AUS, 3: BOASG
         $FLAG[334] = FALSE
      ;ENDFOLD
      ;FOLD -- Quitt. Fraesen SK1 -- ;%{SE}%MKUKATPVW %CVW_COM %VCOMMENT %P 2:-- Quitt. Fraesen SK1 --, 3: VW_COMMENT
      ;ENDFOLD
      ;FOLD A786 = (!F322 & !F830) + (F830 & A786) + (E193 + A3505) & EIN ;%{SE}%MKUKATPVW %CVW_SPS %VBOASG %P 2:A786 = (!F322 & !F830) + (F830 & A786) + (E193 + A3505) & EIN, 3: BOASG
         $OUT[786] = (NOT $FLAG[322] AND NOT $FLAG[830]) OR ($FLAG[830] AND $OUT[786]) OR ($IN[193] OR $OUT[3505]) AND TRUE
      ;ENDFOLD
      ;FOLD A3872 = (!F78 & F79 & !F830) + (F830 & A3872) ;%{SE}%MKUKATPVW %CVW_SPS %VBOASG %P 2:A3872 = (!F78 & F79 & !F830) + (F830 & A3872), 3: BOASG
         $OUT[3872] = (NOT $FLAG[78] AND $FLAG[79] AND NOT $FLAG[830]) OR ($FLAG[830] AND $OUT[3872])
      ;ENDFOLD
      ;FOLD A3512 = (F78 & !F79 & !F830) + (F830 & A3512) ;%{SE}%MKUKATPVW %CVW_SPS %VBOASG %P 2:A3512 = (F78 & !F79 & !F830) + (F830 & A3512), 3: BOASG
         $OUT[3512] = ($FLAG[78] AND NOT $FLAG[79] AND NOT $FLAG[830]) OR ($FLAG[830] AND $OUT[3512])
      ;ENDFOLD
      ;FOLD SCHRITT 123 = A4039 & (!E786 & !E788 & !F830) ;%{SE}%MKUKATPVW %CVW_SPS %VST_CON %P 2:SCHRITT 123 = A4039 & (!E786 & !E788 & !F830), 3: ST_CON
         IF $OUT[4039] AND (NOT $IN[786] AND NOT $IN[788] AND NOT $FLAG[830]) THEN
            PREV_STEP[9] = APP_INT_STEP[9]
            APP_INT_STEP[9] = 123
         ENDIF
      ;ENDFOLD
   ;ENDFOLD
   ;FOLD SCHRITT 123 -- st. RZ1 # Ruecksetzen -- ;%{P}%MKUKATPVW,%CSTEP,%VST_NR,%P 1:SCHRITT, 2:123, 3: st. RZ1 # Ruecksetzen
      ;FOLD ;%{H}
         Case 123
      ;ENDFOLD
      ;FOLD -- Start Init Same AUS -- ;%{SE}%MKUKATPVW %CVW_COM %VCOMMENT %P 2:-- Start Init Same AUS --, 3: VW_COMMENT
      ;ENDFOLD
      ;FOLD A3514 = AUS ;%{SE}%MKUKATPVW %CVW_SPS %VBOASG %P 2:A3514 = AUS, 3: BOASG
         $OUT[3514] = FALSE
      ;ENDFOLD
      ;FOLD -- Start Spot AUS -- ;%{SE}%MKUKATPVW %CVW_COM %VCOMMENT %P 2:-- Start Spot AUS --, 3: VW_COMMENT
      ;ENDFOLD
      ;FOLD A3511 = AUS ;%{SE}%MKUKATPVW %CVW_SPS %VBOASG %P 2:A3511 = AUS, 3: BOASG
         $OUT[3511] = FALSE
      ;ENDFOLD
      ;FOLD -- Start Dress AUS -- ;%{SE}%MKUKATPVW %CVW_COM %VCOMMENT %P 2:-- Start Dress AUS --, 3: VW_COMMENT
      ;ENDFOLD
      ;FOLD A3510 = AUS ;%{SE}%MKUKATPVW %CVW_SPS %VBOASG %P 2:A3510 = AUS, 3: BOASG
         $OUT[3510] = FALSE
      ;ENDFOLD
      ;FOLD -- Start Init New AUS -- ;%{SE}%MKUKATPVW %CVW_COM %VCOMMENT %P 2:-- Start Init New AUS --, 3: VW_COMMENT
      ;ENDFOLD
      ;FOLD A3513 = AUS ;%{SE}%MKUKATPVW %CVW_SPS %VBOASG %P 2:A3513 = AUS, 3: BOASG
         $OUT[3513] = FALSE
      ;ENDFOLD
      ;FOLD -- Start Dress in Position AUS -- ;%{SE}%MKUKATPVW %CVW_COM %VCOMMENT %P 2:-- Start Dress in Position AUS --, 3: VW_COMMENT
      ;ENDFOLD
      ;FOLD A3871 = AUS ;%{SE}%MKUKATPVW %CVW_SPS %VBOASG %P 2:A3871 = AUS, 3: BOASG
         $OUT[3871] = FALSE
      ;ENDFOLD
      ;FOLD -- Start Dress Fin AUS -- ;%{SE}%MKUKATPVW %CVW_COM %VCOMMENT %P 2:-- Start Dress Fin AUS --, 3: VW_COMMENT
      ;ENDFOLD
      ;FOLD A3872 = AUS ;%{SE}%MKUKATPVW %CVW_SPS %VBOASG %P 2:A3872 = AUS, 3: BOASG
         $OUT[3872] = FALSE
      ;ENDFOLD
      ;FOLD -- Start StartAcknowledge AUS -- ;%{SE}%MKUKATPVW %CVW_COM %VCOMMENT %P 2:-- Start StartAcknowledge AUS --, 3: VW_COMMENT
      ;ENDFOLD
      ;FOLD A3512 = AUS ;%{SE}%MKUKATPVW %CVW_SPS %VBOASG %P 2:A3512 = AUS, 3: BOASG
         $OUT[3512] = FALSE
      ;ENDFOLD
      ;FOLD -- Schritt Fraesen aktiv -- ;%{SE}%MKUKATPVW %CVW_COM %VCOMMENT %P 2:-- Schritt Fraesen aktiv --, 3: VW_COMMENT
      ;ENDFOLD
      ;FOLD A3534 = AUS ;%{SE}%MKUKATPVW %CVW_SPS %VBOASG %P 2:A3534 = AUS, 3: BOASG
         $OUT[3534] = FALSE
      ;ENDFOLD
      ;FOLD -- Schritt Messen aktiv -- ;%{SE}%MKUKATPVW %CVW_COM %VCOMMENT %P 2:-- Schritt Messen aktiv --, 3: VW_COMMENT
      ;ENDFOLD
      ;FOLD A3535 = AUS ;%{SE}%MKUKATPVW %CVW_SPS %VBOASG %P 2:A3535 = AUS, 3: BOASG
         $OUT[3535] = FALSE
      ;ENDFOLD
      ;FOLD -- Schritt Schweissen aktiv -- ;%{SE}%MKUKATPVW %CVW_COM %VCOMMENT %P 2:-- Schritt Schweissen aktiv --, 3: VW_COMMENT
      ;ENDFOLD
      ;FOLD A3536 = AUS ;%{SE}%MKUKATPVW %CVW_SPS %VBOASG %P 2:A3536 = AUS, 3: BOASG
         $OUT[3536] = FALSE
      ;ENDFOLD
      ;FOLD -- KF1 Ausblasen AUS -- ;%{SE}%MKUKATPVW %CVW_COM %VCOMMENT %P 2:-- KF1 Ausblasen AUS --, 3: VW_COMMENT
      ;ENDFOLD
      ;FOLD A836 = AUS ;%{SE}%MKUKATPVW %CVW_SPS %VBOASG %P 2:A836 = AUS, 3: BOASG
         $OUT[836] = FALSE
      ;ENDFOLD
      ;FOLD -- Ueberwachungszeit ServoGun SZ1 Messen -- ;%{SE}%MKUKATPVW %CVW_COM %VCOMMENT %P 2:-- Ueberwachungszeit ServoGun SZ1 Messen --, 3: VW_COMMENT
      ;ENDFOLD
      ;FOLD t9 ( EIN ) = -150[1/10Sek] ;%{SE}%MKUKATPVW %CVW_SPS %VTASG %P 2:t9 ( EIN ) = -150[1/10Sek], 3: TASG
         VW(#SET_TIME,TRUE,9,0,-150)
      ;ENDFOLD
      ;FOLD -- Fehler SK ruecksetzen -- ;%{SE}%MKUKATPVW %CVW_COM %VCOMMENT %P 2:-- Fehler SK ruecksetzen --, 3: VW_COMMENT
      ;ENDFOLD
      ;FOLD -- Fehler SK Messen AUS -- ;%{SE}%MKUKATPVW %CVW_COM %VCOMMENT %P 2:-- Fehler SK Messen AUS --, 3: VW_COMMENT
      ;ENDFOLD
      ;FOLD F326 = AUS ;%{SE}%MKUKATPVW %CVW_SPS %VBOASG %P 2:F326 = AUS, 3: BOASG
         $FLAG[326] = FALSE
      ;ENDFOLD
      ;FOLD SCHRITT 124 = A4039 & A3506 & A3505 & A3862 & !E838 ;%{SE}%MKUKATPVW %CVW_SPS %VST_CON %P 2:SCHRITT 124 = A4039 & A3506 & A3505 & A3862 & !E838, 3: ST_CON
         IF $OUT[4039] AND $OUT[3506] AND $OUT[3505] AND $OUT[3862] AND NOT $IN[838] THEN
            PREV_STEP[9] = APP_INT_STEP[9]
            APP_INT_STEP[9] = 124
         ENDIF
      ;ENDFOLD
   ;ENDFOLD
   ;FOLD SCHRITT 124 -- st. RZ1 # Messen -- ;%{P}%MKUKATPVW,%CSTEP,%VST_NR,%P 1:SCHRITT, 2:124, 3: st. RZ1 # Messen
      ;FOLD ;%{H}
         Case 124
      ;ENDFOLD
      ;FOLD -- Kommentar -- ;%{SE}%MKUKATPVW %CVW_COM %VCOMMENT %P 2:-- Kommentar --, 3: VW_COMMENT
      ;ENDFOLD
      ;FOLD -- Messen nach Fraesen -- ;%{SE}%MKUKATPVW %CVW_COM %VCOMMENT %P 2:-- Messen nach Fraesen --, 3: VW_COMMENT
      ;ENDFOLD
      ;FOLD A3514 = EIN ;%{SE}%MKUKATPVW %CVW_SPS %VBOASG %P 2:A3514 = EIN, 3: BOASG
         $OUT[3514] = TRUE
      ;ENDFOLD
      ;FOLD A3510 = EIN ;%{SE}%MKUKATPVW %CVW_SPS %VBOASG %P 2:A3510 = EIN, 3: BOASG
         $OUT[3510] = TRUE
      ;ENDFOLD
      ;FOLD -- Schritt Messen aktiv -- ;%{SE}%MKUKATPVW %CVW_COM %VCOMMENT %P 2:-- Schritt Messen aktiv --, 3: VW_COMMENT
      ;ENDFOLD
      ;FOLD A3535 = EIN ;%{SE}%MKUKATPVW %CVW_SPS %VBOASG %P 2:A3535 = EIN, 3: BOASG
         $OUT[3535] = TRUE
      ;ENDFOLD
      ;FOLD SCHRITT 125 = A4039 ;%{SE}%MKUKATPVW %CVW_SPS %VST_CON %P 2:SCHRITT 125 = A4039, 3: ST_CON
         IF $OUT[4039] THEN
            PREV_STEP[9] = APP_INT_STEP[9]
            APP_INT_STEP[9] = 125
         ENDIF
      ;ENDFOLD
   ;ENDFOLD
   ;FOLD SCHRITT 125 -- st. RZ1 # Auswertung -- ;%{P}%MKUKATPVW,%CSTEP,%VST_NR,%P 1:SCHRITT, 2:125, 3: st. RZ1 # Auswertung
      ;FOLD ;%{H}
         Case 125
      ;ENDFOLD
      ;FOLD -- Auswertung Messung -- ;%{SE}%MKUKATPVW %CVW_COM %VCOMMENT %P 2:-- Auswertung Messung --, 3: VW_COMMENT
      ;ENDFOLD
      ;FOLD SCHRITT 127 = A4039 & A3508 ;%{SE}%MKUKATPVW %CVW_SPS %VST_CON %P 2:SCHRITT 127 = A4039 & A3508, 3: ST_CON
         IF $OUT[4039] AND $OUT[3508] THEN
            PREV_STEP[9] = APP_INT_STEP[9]
            APP_INT_STEP[9] = 127
         ENDIF
      ;ENDFOLD
      ;FOLD SCHRITT 126 = A4039 & A3509 ;%{SE}%MKUKATPVW %CVW_SPS %VST_CON %P 2:SCHRITT 126 = A4039 & A3509, 3: ST_CON
         IF $OUT[4039] AND $OUT[3509] THEN
            PREV_STEP[9] = APP_INT_STEP[9]
            APP_INT_STEP[9] = 126
         ENDIF
      ;ENDFOLD
   ;ENDFOLD
   ;FOLD SCHRITT 126 -- st. RZ1 # Fehler Messen -- ;%{P}%MKUKATPVW,%CSTEP,%VST_NR,%P 1:SCHRITT, 2:126, 3: st. RZ1 # Fehler Messen
      ;FOLD ;%{H}
         Case 126
      ;ENDFOLD
      ;FOLD -- Start Init Same AUS -- ;%{SE}%MKUKATPVW %CVW_COM %VCOMMENT %P 2:-- Start Init Same AUS --, 3: VW_COMMENT
      ;ENDFOLD
      ;FOLD A3514 = AUS ;%{SE}%MKUKATPVW %CVW_SPS %VBOASG %P 2:A3514 = AUS, 3: BOASG
         $OUT[3514] = FALSE
      ;ENDFOLD
      ;FOLD -- Start Spot AUS -- ;%{SE}%MKUKATPVW %CVW_COM %VCOMMENT %P 2:-- Start Spot AUS --, 3: VW_COMMENT
      ;ENDFOLD
      ;FOLD A3511 = AUS ;%{SE}%MKUKATPVW %CVW_SPS %VBOASG %P 2:A3511 = AUS, 3: BOASG
         $OUT[3511] = FALSE
      ;ENDFOLD
      ;FOLD -- Start Dress AUS -- ;%{SE}%MKUKATPVW %CVW_COM %VCOMMENT %P 2:-- Start Dress AUS --, 3: VW_COMMENT
      ;ENDFOLD
      ;FOLD A3510 = AUS ;%{SE}%MKUKATPVW %CVW_SPS %VBOASG %P 2:A3510 = AUS, 3: BOASG
         $OUT[3510] = FALSE
      ;ENDFOLD
      ;FOLD -- Start Init New AUS -- ;%{SE}%MKUKATPVW %CVW_COM %VCOMMENT %P 2:-- Start Init New AUS --, 3: VW_COMMENT
      ;ENDFOLD
      ;FOLD A3513 = AUS ;%{SE}%MKUKATPVW %CVW_SPS %VBOASG %P 2:A3513 = AUS, 3: BOASG
         $OUT[3513] = FALSE
      ;ENDFOLD
      ;FOLD -- Start Dress in Position AUS -- ;%{SE}%MKUKATPVW %CVW_COM %VCOMMENT %P 2:-- Start Dress in Position AUS --, 3: VW_COMMENT
      ;ENDFOLD
      ;FOLD A3871 = AUS ;%{SE}%MKUKATPVW %CVW_SPS %VBOASG %P 2:A3871 = AUS, 3: BOASG
         $OUT[3871] = FALSE
      ;ENDFOLD
      ;FOLD -- Start Dress Fin AUS -- ;%{SE}%MKUKATPVW %CVW_COM %VCOMMENT %P 2:-- Start Dress Fin AUS --, 3: VW_COMMENT
      ;ENDFOLD
      ;FOLD A3872 = AUS ;%{SE}%MKUKATPVW %CVW_SPS %VBOASG %P 2:A3872 = AUS, 3: BOASG
         $OUT[3872] = FALSE
      ;ENDFOLD
      ;FOLD -- Start StartAcknowledge AUS -- ;%{SE}%MKUKATPVW %CVW_COM %VCOMMENT %P 2:-- Start StartAcknowledge AUS --, 3: VW_COMMENT
      ;ENDFOLD
      ;FOLD A3512 = AUS ;%{SE}%MKUKATPVW %CVW_SPS %VBOASG %P 2:A3512 = AUS, 3: BOASG
         $OUT[3512] = FALSE
      ;ENDFOLD
      ;FOLD -- Kommentar -- ;%{SE}%MKUKATPVW %CVW_COM %VCOMMENT %P 2:-- Kommentar --, 3: VW_COMMENT
      ;ENDFOLD
      ;FOLD -- RSK Sammelstoerung -- ;%{SE}%MKUKATPVW %CVW_COM %VCOMMENT %P 2:-- RSK Sammelstoerung --, 3: VW_COMMENT
      ;ENDFOLD
      ;FOLD F326 = EIN ;%{SE}%MKUKATPVW %CVW_SPS %VBOASG %P 2:F326 = EIN, 3: BOASG
         $FLAG[326] = TRUE
      ;ENDFOLD
      ;FOLD F329 = F326 ;%{SE}%MKUKATPVW %CVW_SPS %VBOASG %P 2:F329 = F326, 3: BOASG
         $FLAG[329] = $FLAG[326]
      ;ENDFOLD
      ;FOLD -- Flagbildung Wiederholfraesen -- ;%{SE}%MKUKATPVW %CVW_COM %VCOMMENT %P 2:-- Flagbildung Wiederholfraesen --, 3: VW_COMMENT
      ;ENDFOLD
      ;FOLD F749 = (F322 + F323 + F325 + F326 + F327 + F329) & !F748 ;%{SE}%MKUKATPVW %CVW_SPS %VBOASG %P 2:F749 = (F322 + F323 + F325 + F326 + F327 + F329) & !F748, 3: BOASG
         $FLAG[749] = ($FLAG[322] OR $FLAG[323] OR $FLAG[325] OR $FLAG[326] OR $FLAG[327] OR $FLAG[329]) AND NOT $FLAG[748]
      ;ENDFOLD
      ;FOLD SCHRITT 123 = A4039 & F326 & F329 & A3862 & (E26 + E27) ;%{SE}%MKUKATPVW %CVW_SPS %VST_CON %P 2:SCHRITT 123 = A4039 & F326 & F329 & A3862 & (E26 + E27), 3: ST_CON
         IF $OUT[4039] AND $FLAG[326] AND $FLAG[329] AND $OUT[3862] AND ($IN[26] OR $IN[27]) THEN
            PREV_STEP[9] = APP_INT_STEP[9]
            APP_INT_STEP[9] = 123
         ENDIF
      ;ENDFOLD
      ;FOLD SCHRITT 150 = A4039 & F326 & F329 & A3862 & A140 ;%{SE}%MKUKATPVW %CVW_SPS %VST_CON %P 2:SCHRITT 150 = A4039 & F326 & F329 & A3862 & A140, 3: ST_CON
         IF $OUT[4039] AND $FLAG[326] AND $FLAG[329] AND $OUT[3862] AND $OUT[140] THEN
            PREV_STEP[9] = APP_INT_STEP[9]
            APP_INT_STEP[9] = 150
         ENDIF
      ;ENDFOLD
   ;ENDFOLD
   ;FOLD SCHRITT 127 -- st. RZ1 # Acknowledge -- ;%{P}%MKUKATPVW,%CSTEP,%VST_NR,%P 1:SCHRITT, 2:127, 3: st. RZ1 # Acknowledge
      ;FOLD ;%{H}
         Case 127
      ;ENDFOLD
      ;FOLD -- ServoGun - StartAcknowledge -- ;%{SE}%MKUKATPVW %CVW_COM %VCOMMENT %P 2:-- ServoGun - StartAcknowledge --, 3: VW_COMMENT
      ;ENDFOLD
      ;FOLD -- Start Dress AUS -- ;%{SE}%MKUKATPVW %CVW_COM %VCOMMENT %P 2:-- Start Dress AUS --, 3: VW_COMMENT
      ;ENDFOLD
      ;FOLD A3510 = AUS ;%{SE}%MKUKATPVW %CVW_SPS %VBOASG %P 2:A3510 = AUS, 3: BOASG
         $OUT[3510] = FALSE
      ;ENDFOLD
      ;FOLD -- Start Init Same AUS -- ;%{SE}%MKUKATPVW %CVW_COM %VCOMMENT %P 2:-- Start Init Same AUS --, 3: VW_COMMENT
      ;ENDFOLD
      ;FOLD A3514 = AUS ;%{SE}%MKUKATPVW %CVW_SPS %VBOASG %P 2:A3514 = AUS, 3: BOASG
         $OUT[3514] = FALSE
      ;ENDFOLD
      ;FOLD -- Start StartAcknowledge EIN -- ;%{SE}%MKUKATPVW %CVW_COM %VCOMMENT %P 2:-- Start StartAcknowledge EIN --, 3: VW_COMMENT
      ;ENDFOLD
      ;FOLD A3512 = EIN ;%{SE}%MKUKATPVW %CVW_SPS %VBOASG %P 2:A3512 = EIN, 3: BOASG
         $OUT[3512] = TRUE
      ;ENDFOLD
      ;FOLD -- Schritt Messen aktiv -- ;%{SE}%MKUKATPVW %CVW_COM %VCOMMENT %P 2:-- Schritt Messen aktiv --, 3: VW_COMMENT
      ;ENDFOLD
      ;FOLD A3535 = AUS ;%{SE}%MKUKATPVW %CVW_SPS %VBOASG %P 2:A3535 = AUS, 3: BOASG
         $OUT[3535] = FALSE
      ;ENDFOLD
      ;FOLD SCHRITT 129 = !F335 & A4039 & !A3507 ;%{SE}%MKUKATPVW %CVW_SPS %VST_CON %P 2:SCHRITT 129 = !F335 & A4039 & !A3507, 3: ST_CON
         IF NOT $FLAG[335] AND $OUT[4039] AND NOT $OUT[3507] THEN
            PREV_STEP[9] = APP_INT_STEP[9]
            APP_INT_STEP[9] = 129
         ENDIF
      ;ENDFOLD
      ;FOLD SCHRITT 129 = F335 & !F78 & A4039 & !A3507 ;%{SE}%MKUKATPVW %CVW_SPS %VST_CON %P 2:SCHRITT 129 = F335 & !F78 & A4039 & !A3507, 3: ST_CON
         IF $FLAG[335] AND NOT $FLAG[78] AND $OUT[4039] AND NOT $OUT[3507] THEN
            PREV_STEP[9] = APP_INT_STEP[9]
            APP_INT_STEP[9] = 129
         ENDIF
      ;ENDFOLD
      ;FOLD Schritt 190 = F335 & F78 & A4039 & !A3507 ;%{SE}%MKUKATPVW %CVW_SPS %VST_CON %P 2:Schritt 190 = F335 & F78 & A4039 & !A3507, 3: ST_CON
         IF $FLAG[335] AND $FLAG[78] AND $OUT[4039] AND NOT $OUT[3507] THEN
            PREV_STEP[9] = APP_INT_STEP[9]
            APP_INT_STEP[9] = 190
         ENDIF
      ;ENDFOLD
   ;ENDFOLD
   ;FOLD SCHRITT 129 -- st. RZ1 # Ruecksetzen -- ;%{P}%MKUKATPVW,%CSTEP,%VST_NR,%P 1:SCHRITT, 2:129, 3: st. RZ1 # Ruecksetzen
      ;FOLD ;%{H}
         Case 129
      ;ENDFOLD
      ;FOLD -- Start Init Same AUS -- ;%{SE}%MKUKATPVW %CVW_COM %VCOMMENT %P 2:-- Start Init Same AUS --, 3: VW_COMMENT
      ;ENDFOLD
      ;FOLD A3514 = AUS ;%{SE}%MKUKATPVW %CVW_SPS %VBOASG %P 2:A3514 = AUS, 3: BOASG
         $OUT[3514] = FALSE
      ;ENDFOLD
      ;FOLD -- Start Spot AUS -- ;%{SE}%MKUKATPVW %CVW_COM %VCOMMENT %P 2:-- Start Spot AUS --, 3: VW_COMMENT
      ;ENDFOLD
      ;FOLD A3511 = AUS ;%{SE}%MKUKATPVW %CVW_SPS %VBOASG %P 2:A3511 = AUS, 3: BOASG
         $OUT[3511] = FALSE
      ;ENDFOLD
      ;FOLD -- Start Dress AUS -- ;%{SE}%MKUKATPVW %CVW_COM %VCOMMENT %P 2:-- Start Dress AUS --, 3: VW_COMMENT
      ;ENDFOLD
      ;FOLD A3510 = AUS ;%{SE}%MKUKATPVW %CVW_SPS %VBOASG %P 2:A3510 = AUS, 3: BOASG
         $OUT[3510] = FALSE
      ;ENDFOLD
      ;FOLD -- Start Init New AUS -- ;%{SE}%MKUKATPVW %CVW_COM %VCOMMENT %P 2:-- Start Init New AUS --, 3: VW_COMMENT
      ;ENDFOLD
      ;FOLD A3513 = AUS ;%{SE}%MKUKATPVW %CVW_SPS %VBOASG %P 2:A3513 = AUS, 3: BOASG
         $OUT[3513] = FALSE
      ;ENDFOLD
      ;FOLD -- Start Dress in Position AUS -- ;%{SE}%MKUKATPVW %CVW_COM %VCOMMENT %P 2:-- Start Dress in Position AUS --, 3: VW_COMMENT
      ;ENDFOLD
      ;FOLD A3871 = AUS ;%{SE}%MKUKATPVW %CVW_SPS %VBOASG %P 2:A3871 = AUS, 3: BOASG
         $OUT[3871] = FALSE
      ;ENDFOLD
      ;FOLD -- Start Dress Fin AUS -- ;%{SE}%MKUKATPVW %CVW_COM %VCOMMENT %P 2:-- Start Dress Fin AUS --, 3: VW_COMMENT
      ;ENDFOLD
      ;FOLD A3872 = AUS ;%{SE}%MKUKATPVW %CVW_SPS %VBOASG %P 2:A3872 = AUS, 3: BOASG
         $OUT[3872] = FALSE
      ;ENDFOLD
      ;FOLD -- Start StartAcknowledge AUS -- ;%{SE}%MKUKATPVW %CVW_COM %VCOMMENT %P 2:-- Start StartAcknowledge AUS --, 3: VW_COMMENT
      ;ENDFOLD
      ;FOLD A3512 = AUS ;%{SE}%MKUKATPVW %CVW_SPS %VBOASG %P 2:A3512 = AUS, 3: BOASG
         $OUT[3512] = FALSE
      ;ENDFOLD
      ;FOLD bin30 ( EIN ) = 0 ;%{SE}%MKUKATPVW %CVW_SPS %VARIASG %P 2:bin30 ( EIN ) = 0, 3: ARIASG
         VW(#BINOUT,TRUE,30,0)
      ;ENDFOLD
      ;FOLD -- Schritt Fraesen aktiv -- ;%{SE}%MKUKATPVW %CVW_COM %VCOMMENT %P 2:-- Schritt Fraesen aktiv --, 3: VW_COMMENT
      ;ENDFOLD
      ;FOLD A3534 = AUS ;%{SE}%MKUKATPVW %CVW_SPS %VBOASG %P 2:A3534 = AUS, 3: BOASG
         $OUT[3534] = FALSE
      ;ENDFOLD
      ;FOLD -- Schritt Messen aktiv -- ;%{SE}%MKUKATPVW %CVW_COM %VCOMMENT %P 2:-- Schritt Messen aktiv --, 3: VW_COMMENT
      ;ENDFOLD
      ;FOLD A3535 = AUS ;%{SE}%MKUKATPVW %CVW_SPS %VBOASG %P 2:A3535 = AUS, 3: BOASG
         $OUT[3535] = FALSE
      ;ENDFOLD
      ;FOLD -- Schritt Schweissen aktiv -- ;%{SE}%MKUKATPVW %CVW_COM %VCOMMENT %P 2:-- Schritt Schweissen aktiv --, 3: VW_COMMENT
      ;ENDFOLD
      ;FOLD A3536 = AUS ;%{SE}%MKUKATPVW %CVW_SPS %VBOASG %P 2:A3536 = AUS, 3: BOASG
         $OUT[3536] = FALSE
      ;ENDFOLD
      ;FOLD -- Fehler SK ruecksetzen -- ;%{SE}%MKUKATPVW %CVW_COM %VCOMMENT %P 2:-- Fehler SK ruecksetzen --, 3: VW_COMMENT
      ;ENDFOLD
      ;FOLD -- Druckvorgabe SK1/ServoGun -- ;%{SE}%MKUKATPVW %CVW_COM %VCOMMENT %P 2:-- Druckvorgabe SK1/ServoGun --, 3: VW_COMMENT
      ;ENDFOLD
      ;FOLD bin1 ( F78 ) = 41 ;%{SE}%MKUKATPVW %CVW_SPS %VARIASG %P 2:bin1 ( F78 ) = 41, 3: ARIASG
         VW(#BINOUT,$FLAG[78],1,41)
      ;ENDFOLD
      ;FOLD bin1 ( F79 ) = 51 ;%{SE}%MKUKATPVW %CVW_SPS %VARIASG %P 2:bin1 ( F79 ) = 51, 3: ARIASG
         VW(#BINOUT,$FLAG[79],1,51)
      ;ENDFOLD
      ;FOLD bin31 ( F78 ) = 41 ;%{SE}%MKUKATPVW %CVW_SPS %VARIASG %P 2:bin31 ( F78 ) = 41, 3: ARIASG
         VW(#BINOUT,$FLAG[78],31,41)
      ;ENDFOLD
      ;FOLD bin31 ( F79 ) = 51 ;%{SE}%MKUKATPVW %CVW_SPS %VARIASG %P 2:bin31 ( F79 ) = 51, 3: ARIASG
         VW(#BINOUT,$FLAG[79],31,51)
      ;ENDFOLD
      ;FOLD -- Wartezeit Programmwechsel SK -- ;%{SE}%MKUKATPVW %CVW_COM %VCOMMENT %P 2:-- Wartezeit Programmwechsel SK --, 3: VW_COMMENT
      ;ENDFOLD
      ;FOLD T8 ( !F334 ) = -2[1/10Sek] ;%{SE}%MKUKATPVW %CVW_SPS %VTASG %P 2:T8 ( !F334 ) = -2[1/10Sek], 3: TASG
         VW(#SET_TIME,NOT $FLAG[334],8,0,-2)
      ;ENDFOLD
      ;FOLD -- Hilfsflag SK Programmwechsel -- ;%{SE}%MKUKATPVW %CVW_COM %VCOMMENT %P 2:-- Hilfsflag SK Programmwechsel --, 3: VW_COMMENT
      ;ENDFOLD
      ;FOLD F334 = EIN ;%{SE}%MKUKATPVW %CVW_SPS %VBOASG %P 2:F334 = EIN, 3: BOASG
         $FLAG[334] = TRUE
      ;ENDFOLD
      ;FOLD t9 ( EIN ) = STOP ;%{SE}%MKUKATPVW %CVW_SPS %VTSTOP %P 2:t9 ( EIN ) = STOP, 3: TSTOP
         VW(#SET_TIME,TRUE,9,1,0)
      ;ENDFOLD
      ;FOLD SCHRITT 130 = T8 & A4039 & A3506 & A3505 & A3862 & !E838 ;%{SE}%MKUKATPVW %CVW_SPS %VST_CON %P 2:SCHRITT 130 = T8 & A4039 & A3506 & A3505 & A3862 & !E838, 3: ST_CON
         IF $TIMER_FLAG[8] AND $OUT[4039] AND $OUT[3506] AND $OUT[3505] AND $OUT[3862] AND NOT $IN[838] THEN
            PREV_STEP[9] = APP_INT_STEP[9]
            APP_INT_STEP[9] = 130
         ENDIF
      ;ENDFOLD
   ;ENDFOLD
   ;FOLD SCHRITT 130 -- st. RZ1 # Schweissen -- ;%{P}%MKUKATPVW,%CSTEP,%VST_NR,%P 1:SCHRITT, 2:130, 3: st. RZ1 # Schweissen
      ;FOLD ;%{H}
         Case 130
      ;ENDFOLD
      ;FOLD -- Schritt Schweissen aktiv -- ;%{SE}%MKUKATPVW %CVW_COM %VCOMMENT %P 2:-- Schritt Schweissen aktiv --, 3: VW_COMMENT
      ;ENDFOLD
      ;FOLD A3536 = EIN ;%{SE}%MKUKATPVW %CVW_SPS %VBOASG %P 2:A3536 = EIN, 3: BOASG
         $OUT[3536] = TRUE
      ;ENDFOLD
      ;FOLD -- Hilfsflag SK Programmwechsel -- ;%{SE}%MKUKATPVW %CVW_COM %VCOMMENT %P 2:-- Hilfsflag SK Programmwechsel --, 3: VW_COMMENT
      ;ENDFOLD
      ;FOLD F334 = AUS ;%{SE}%MKUKATPVW %CVW_SPS %VBOASG %P 2:F334 = AUS, 3: BOASG
         $FLAG[334] = FALSE
      ;ENDFOLD
      ;FOLD A3518 = A3519 ;%{SE}%MKUKATPVW %CVW_SPS %VBOASG %P 2:A3518 = A3519, 3: BOASG
         $OUT[3518] = $OUT[3519]
      ;ENDFOLD
      ;FOLD F748 = A3518 ;%{SE}%MKUKATPVW %CVW_SPS %VBOASG %P 2:F748 = A3518, 3: BOASG
         $FLAG[748] = $OUT[3518]
      ;ENDFOLD
      ;FOLD -- Schritt Schweissen aktiv -- ;%{SE}%MKUKATPVW %CVW_COM %VCOMMENT %P 2:-- Schritt Schweissen aktiv --, 3: VW_COMMENT
      ;ENDFOLD
      ;FOLD A3536 = EIN ;%{SE}%MKUKATPVW %CVW_SPS %VBOASG %P 2:A3536 = EIN, 3: BOASG
         $OUT[3536] = TRUE
      ;ENDFOLD
      ;FOLD -- ServoGun - Start Spot EIN -- ;%{SE}%MKUKATPVW %CVW_COM %VCOMMENT %P 2:-- ServoGun - Start Spot EIN --, 3: VW_COMMENT
      ;ENDFOLD
      ;FOLD A3511 = EIN ;%{SE}%MKUKATPVW %CVW_SPS %VBOASG %P 2:A3511 = EIN, 3: BOASG
         $OUT[3511] = TRUE
      ;ENDFOLD
      ;FOLD F749 = AUS ;%{SE}%MKUKATPVW %CVW_SPS %VBOASG %P 2:F749 = AUS, 3: BOASG
         $FLAG[749] = FALSE
      ;ENDFOLD
      ;FOLD SCHRITT 131 = A4039 ;%{SE}%MKUKATPVW %CVW_SPS %VST_CON %P 2:SCHRITT 131 = A4039, 3: ST_CON
         IF $OUT[4039] THEN
            PREV_STEP[9] = APP_INT_STEP[9]
            APP_INT_STEP[9] = 131
         ENDIF
      ;ENDFOLD
   ;ENDFOLD
   ;FOLD SCHRITT 131 -- st. RZ1 # Auswertung -- ;%{P}%MKUKATPVW,%CSTEP,%VST_NR,%P 1:SCHRITT, 2:131, 3: st. RZ1 # Auswertung
      ;FOLD ;%{H}
         Case 131
      ;ENDFOLD
      ;FOLD -- Auswertung -- ;%{SE}%MKUKATPVW %CVW_COM %VCOMMENT %P 2:-- Auswertung --, 3: VW_COMMENT
      ;ENDFOLD
      ;FOLD Schritt 132 = A3509 & !E804 & E805 ;%{SE}%MKUKATPVW %CVW_SPS %VST_CON %P 2:Schritt 132 = A3509 & !E804 & E805, 3: ST_CON
         IF $OUT[3509] AND NOT $IN[804] AND $IN[805] THEN
            PREV_STEP[9] = APP_INT_STEP[9]
            APP_INT_STEP[9] = 132
         ENDIF
      ;ENDFOLD
      ;FOLD SCHRITT 133 = A3508 & (E804 & !E806 + !A785 & E15) ;%{SE}%MKUKATPVW %CVW_SPS %VST_CON %P 2:SCHRITT 133 = A3508 & (E804 & !E806 + !A785 & E15), 3: ST_CON
         IF $OUT[3508] AND ($IN[804] AND NOT $IN[806] OR NOT $OUT[785] AND $IN[15]) THEN
            PREV_STEP[9] = APP_INT_STEP[9]
            APP_INT_STEP[9] = 133
         ENDIF
      ;ENDFOLD
   ;ENDFOLD
   ;FOLD SCHRITT 132 -- st. RZ1 # Fehler Schweissung -- ;%{P}%MKUKATPVW,%CSTEP,%VST_NR,%P 1:SCHRITT, 2:132, 3: st. RZ1 # Fehler Schweissung
      ;FOLD ;%{H}
         Case 132
      ;ENDFOLD
      ;FOLD -- Start Init Same AUS -- ;%{SE}%MKUKATPVW %CVW_COM %VCOMMENT %P 2:-- Start Init Same AUS --, 3: VW_COMMENT
      ;ENDFOLD
      ;FOLD A3514 = AUS ;%{SE}%MKUKATPVW %CVW_SPS %VBOASG %P 2:A3514 = AUS, 3: BOASG
         $OUT[3514] = FALSE
      ;ENDFOLD
      ;FOLD -- Start Spot AUS -- ;%{SE}%MKUKATPVW %CVW_COM %VCOMMENT %P 2:-- Start Spot AUS --, 3: VW_COMMENT
      ;ENDFOLD
      ;FOLD A3511 = AUS ;%{SE}%MKUKATPVW %CVW_SPS %VBOASG %P 2:A3511 = AUS, 3: BOASG
         $OUT[3511] = FALSE
      ;ENDFOLD
      ;FOLD -- Start Dress AUS -- ;%{SE}%MKUKATPVW %CVW_COM %VCOMMENT %P 2:-- Start Dress AUS --, 3: VW_COMMENT
      ;ENDFOLD
      ;FOLD A3510 = AUS ;%{SE}%MKUKATPVW %CVW_SPS %VBOASG %P 2:A3510 = AUS, 3: BOASG
         $OUT[3510] = FALSE
      ;ENDFOLD
      ;FOLD -- Start Init New AUS -- ;%{SE}%MKUKATPVW %CVW_COM %VCOMMENT %P 2:-- Start Init New AUS --, 3: VW_COMMENT
      ;ENDFOLD
      ;FOLD A3513 = AUS ;%{SE}%MKUKATPVW %CVW_SPS %VBOASG %P 2:A3513 = AUS, 3: BOASG
         $OUT[3513] = FALSE
      ;ENDFOLD
      ;FOLD -- Start Dress in Position AUS -- ;%{SE}%MKUKATPVW %CVW_COM %VCOMMENT %P 2:-- Start Dress in Position AUS --, 3: VW_COMMENT
      ;ENDFOLD
      ;FOLD A3871 = AUS ;%{SE}%MKUKATPVW %CVW_SPS %VBOASG %P 2:A3871 = AUS, 3: BOASG
         $OUT[3871] = FALSE
      ;ENDFOLD
      ;FOLD -- Start Dress Fin AUS -- ;%{SE}%MKUKATPVW %CVW_COM %VCOMMENT %P 2:-- Start Dress Fin AUS --, 3: VW_COMMENT
      ;ENDFOLD
      ;FOLD A3872 = AUS ;%{SE}%MKUKATPVW %CVW_SPS %VBOASG %P 2:A3872 = AUS, 3: BOASG
         $OUT[3872] = FALSE
      ;ENDFOLD
      ;FOLD -- Start StartAcknowledge AUS -- ;%{SE}%MKUKATPVW %CVW_COM %VCOMMENT %P 2:-- Start StartAcknowledge AUS --, 3: VW_COMMENT
      ;ENDFOLD
      ;FOLD A3512 = AUS ;%{SE}%MKUKATPVW %CVW_SPS %VBOASG %P 2:A3512 = AUS, 3: BOASG
         $OUT[3512] = FALSE
      ;ENDFOLD
      ;FOLD -- RSK Fehlerausgabe Kraftaufbau -- ;%{SE}%MKUKATPVW %CVW_COM %VCOMMENT %P 2:-- RSK Fehlerausgabe Kraftaufbau --, 3: VW_COMMENT
      ;ENDFOLD
      ;FOLD F325 = AUS ;%{SE}%MKUKATPVW %CVW_SPS %VBOASG %P 2:F325 = AUS, 3: BOASG
         $FLAG[325] = FALSE
      ;ENDFOLD
      ;FOLD -- RSK Fehlerausgabe -- ;%{SE}%MKUKATPVW %CVW_COM %VCOMMENT %P 2:-- RSK Fehlerausgabe --, 3: VW_COMMENT
      ;ENDFOLD
      ;FOLD F327 = EIN ;%{SE}%MKUKATPVW %CVW_SPS %VBOASG %P 2:F327 = EIN, 3: BOASG
         $FLAG[327] = TRUE
      ;ENDFOLD
      ;FOLD F78 = !F327 & F78 ;%{SE}%MKUKATPVW %CVW_SPS %VBOASG %P 2:F78 = !F327 & F78, 3: BOASG
         $FLAG[78] = NOT $FLAG[327] AND $FLAG[78]
      ;ENDFOLD
      ;FOLD F79 = F327 + F79 ;%{SE}%MKUKATPVW %CVW_SPS %VBOASG %P 2:F79 = F327 + F79, 3: BOASG
         $FLAG[79] = $FLAG[327] OR $FLAG[79]
      ;ENDFOLD
      ;FOLD -- RSK Sammelstoerung -- ;%{SE}%MKUKATPVW %CVW_COM %VCOMMENT %P 2:-- RSK Sammelstoerung --, 3: VW_COMMENT
      ;ENDFOLD
      ;FOLD F329 = F325 + F326 + F327 ;%{SE}%MKUKATPVW %CVW_SPS %VBOASG %P 2:F329 = F325 + F326 + F327, 3: BOASG
         $FLAG[329] = $FLAG[325] OR $FLAG[326] OR $FLAG[327]
      ;ENDFOLD
      ;FOLD A3519 = EIN ;%{SE}%MKUKATPVW %CVW_SPS %VBOASG %P 2:A3519 = EIN, 3: BOASG
         $OUT[3519] = TRUE
      ;ENDFOLD
      ;FOLD -- Flagbildung Wiederholfraesen -- ;%{SE}%MKUKATPVW %CVW_COM %VCOMMENT %P 2:-- Flagbildung Wiederholfraesen --, 3: VW_COMMENT
      ;ENDFOLD
      ;FOLD F749 = F329 & !A3518 ;%{SE}%MKUKATPVW %CVW_SPS %VBOASG %P 2:F749 = F329 & !A3518, 3: BOASG
         $FLAG[749] = $FLAG[329] AND NOT $OUT[3518]
      ;ENDFOLD
      ;FOLD A144 = A3518 ;%{SE}%MKUKATPVW %CVW_SPS %VBOASG %P 2:A144 = A3518, 3: BOASG
         $OUT[144] = $OUT[3518]
      ;ENDFOLD
      ;FOLD Schritt 165 = A3862 & A3518 ;%{SE}%MKUKATPVW %CVW_SPS %VST_CON %P 2:Schritt 165 = A3862 & A3518, 3: ST_CON
         IF $OUT[3862] AND $OUT[3518] THEN
            PREV_STEP[9] = APP_INT_STEP[9]
            APP_INT_STEP[9] = 165
         ENDIF
      ;ENDFOLD
      ;FOLD Schritt 103 = A3862 & !A3518 & F749 & A4039 ;%{SE}%MKUKATPVW %CVW_SPS %VST_CON %P 2:Schritt 103 = A3862 & !A3518 & F749 & A4039, 3: ST_CON
         IF $OUT[3862] AND NOT $OUT[3518] AND $FLAG[749] AND $OUT[4039] THEN
            PREV_STEP[9] = APP_INT_STEP[9]
            APP_INT_STEP[9] = 103
         ENDIF
      ;ENDFOLD
   ;ENDFOLD
   ;FOLD SCHRITT 133 -- st. RZ1 # Acknowledge -- ;%{P}%MKUKATPVW,%CSTEP,%VST_NR,%P 1:SCHRITT, 2:133, 3: st. RZ1 # Acknowledge
      ;FOLD ;%{H}
         Case 133
      ;ENDFOLD
      ;FOLD -- ServoGun SZ1 oeffnen -- ;%{SE}%MKUKATPVW %CVW_COM %VCOMMENT %P 2:-- ServoGun SZ1 oeffnen --, 3: VW_COMMENT
      ;ENDFOLD
      ;FOLD A3511 = AUS ;%{SE}%MKUKATPVW %CVW_SPS %VBOASG %P 2:A3511 = AUS, 3: BOASG
         $OUT[3511] = FALSE
      ;ENDFOLD
      ;FOLD A3512 = EIN ;%{SE}%MKUKATPVW %CVW_SPS %VBOASG %P 2:A3512 = EIN, 3: BOASG
         $OUT[3512] = TRUE
      ;ENDFOLD
      ;FOLD -- RSK Fehlerausgabe Kraftaufbau -- ;%{SE}%MKUKATPVW %CVW_COM %VCOMMENT %P 2:-- RSK Fehlerausgabe Kraftaufbau --, 3: VW_COMMENT
      ;ENDFOLD
      ;FOLD F325 = AUS ;%{SE}%MKUKATPVW %CVW_SPS %VBOASG %P 2:F325 = AUS, 3: BOASG
         $FLAG[325] = FALSE
      ;ENDFOLD
      ;FOLD -- RSK Fehlerausgabe -- ;%{SE}%MKUKATPVW %CVW_COM %VCOMMENT %P 2:-- RSK Fehlerausgabe --, 3: VW_COMMENT
      ;ENDFOLD
      ;FOLD F327 = AUS ;%{SE}%MKUKATPVW %CVW_SPS %VBOASG %P 2:F327 = AUS, 3: BOASG
         $FLAG[327] = FALSE
      ;ENDFOLD
      ;FOLD -- RSK Fehlerausgabe -- ;%{SE}%MKUKATPVW %CVW_COM %VCOMMENT %P 2:-- RSK Fehlerausgabe --, 3: VW_COMMENT
      ;ENDFOLD
      ;FOLD F329 = AUS ;%{SE}%MKUKATPVW %CVW_SPS %VBOASG %P 2:F329 = AUS, 3: BOASG
         $FLAG[329] = FALSE
      ;ENDFOLD
      ;FOLD Schritt 134 = A3862 & A3506 & A3505 & !A3507 & A4039 ;%{SE}%MKUKATPVW %CVW_SPS %VST_CON %P 2:Schritt 134 = A3862 & A3506 & A3505 & !A3507 & A4039, 3: ST_CON
         IF $OUT[3862] AND $OUT[3506] AND $OUT[3505] AND NOT $OUT[3507] AND $OUT[4039] THEN
            PREV_STEP[9] = APP_INT_STEP[9]
            APP_INT_STEP[9] = 134
         ENDIF
      ;ENDFOLD
   ;ENDFOLD
   ;FOLD SCHRITT 134 -- st. RZ1 # Ende -- ;%{P}%MKUKATPVW,%CSTEP,%VST_NR,%P 1:SCHRITT, 2:134, 3: st. RZ1 # Ende
      ;FOLD ;%{H}
         Case 134
      ;ENDFOLD
      ;FOLD -- Hilfsflag SK Programmwechsel -- ;%{SE}%MKUKATPVW %CVW_COM %VCOMMENT %P 2:-- Hilfsflag SK Programmwechsel --, 3: VW_COMMENT
      ;ENDFOLD
      ;FOLD F334 = AUS ;%{SE}%MKUKATPVW %CVW_SPS %VBOASG %P 2:F334 = AUS, 3: BOASG
         $FLAG[334] = FALSE
      ;ENDFOLD
      ;FOLD A116 = AUS ;%{SE}%MKUKATPVW %CVW_SPS %VBOASG %P 2:A116 = AUS, 3: BOASG
         $OUT[116] = FALSE
      ;ENDFOLD
      ;FOLD A130 = AUS ;%{SE}%MKUKATPVW %CVW_SPS %VBOASG %P 2:A130 = AUS, 3: BOASG
         $OUT[130] = FALSE
      ;ENDFOLD
      ;FOLD A787 = AUS ;%{SE}%MKUKATPVW %CVW_SPS %VBOASG %P 2:A787 = AUS, 3: BOASG
         $OUT[787] = FALSE
      ;ENDFOLD
      ;FOLD F836 = AUS ;%{SE}%MKUKATPVW %CVW_SPS %VBOASG %P 2:F836 = AUS, 3: BOASG
         $FLAG[836] = FALSE
      ;ENDFOLD
      ;FOLD A140 = AUS ;%{SE}%MKUKATPVW %CVW_SPS %VBOASG %P 2:A140 = AUS, 3: BOASG
         $OUT[140] = FALSE
      ;ENDFOLD
      ;FOLD A144 = AUS ;%{SE}%MKUKATPVW %CVW_SPS %VBOASG %P 2:A144 = AUS, 3: BOASG
         $OUT[144] = FALSE
      ;ENDFOLD
      ;FOLD A150 = AUS ;%{SE}%MKUKATPVW %CVW_SPS %VBOASG %P 2:A150 = AUS, 3: BOASG
         $OUT[150] = FALSE
      ;ENDFOLD
      ;FOLD A3518 = AUS ;%{SE}%MKUKATPVW %CVW_SPS %VBOASG %P 2:A3518 = AUS, 3: BOASG
         $OUT[3518] = FALSE
      ;ENDFOLD
      ;FOLD A3519 = AUS ;%{SE}%MKUKATPVW %CVW_SPS %VBOASG %P 2:A3519 = AUS, 3: BOASG
         $OUT[3519] = FALSE
      ;ENDFOLD
      ;FOLD A3533 = AUS ;%{SE}%MKUKATPVW %CVW_SPS %VBOASG %P 2:A3533 = AUS, 3: BOASG
         $OUT[3533] = FALSE
      ;ENDFOLD
      ;FOLD F748 = AUS ;%{SE}%MKUKATPVW %CVW_SPS %VBOASG %P 2:F748 = AUS, 3: BOASG
         $FLAG[748] = FALSE
      ;ENDFOLD
      ;FOLD F836 = AUS ;%{SE}%MKUKATPVW %CVW_SPS %VBOASG %P 2:F836 = AUS, 3: BOASG
         $FLAG[836] = FALSE
      ;ENDFOLD
      ;FOLD -- Start Init Same AUS -- ;%{SE}%MKUKATPVW %CVW_COM %VCOMMENT %P 2:-- Start Init Same AUS --, 3: VW_COMMENT
      ;ENDFOLD
      ;FOLD A3514 = AUS ;%{SE}%MKUKATPVW %CVW_SPS %VBOASG %P 2:A3514 = AUS, 3: BOASG
         $OUT[3514] = FALSE
      ;ENDFOLD
      ;FOLD -- Start Spot AUS -- ;%{SE}%MKUKATPVW %CVW_COM %VCOMMENT %P 2:-- Start Spot AUS --, 3: VW_COMMENT
      ;ENDFOLD
      ;FOLD A3511 = AUS ;%{SE}%MKUKATPVW %CVW_SPS %VBOASG %P 2:A3511 = AUS, 3: BOASG
         $OUT[3511] = FALSE
      ;ENDFOLD
      ;FOLD -- Start Dress AUS -- ;%{SE}%MKUKATPVW %CVW_COM %VCOMMENT %P 2:-- Start Dress AUS --, 3: VW_COMMENT
      ;ENDFOLD
      ;FOLD A3510 = AUS ;%{SE}%MKUKATPVW %CVW_SPS %VBOASG %P 2:A3510 = AUS, 3: BOASG
         $OUT[3510] = FALSE
      ;ENDFOLD
      ;FOLD -- Start Init New AUS -- ;%{SE}%MKUKATPVW %CVW_COM %VCOMMENT %P 2:-- Start Init New AUS --, 3: VW_COMMENT
      ;ENDFOLD
      ;FOLD A3513 = AUS ;%{SE}%MKUKATPVW %CVW_SPS %VBOASG %P 2:A3513 = AUS, 3: BOASG
         $OUT[3513] = FALSE
      ;ENDFOLD
      ;FOLD -- Dress in Position AUS -- ;%{SE}%MKUKATPVW %CVW_COM %VCOMMENT %P 2:-- Dress in Position AUS --, 3: VW_COMMENT
      ;ENDFOLD
      ;FOLD A3871 = AUS ;%{SE}%MKUKATPVW %CVW_SPS %VBOASG %P 2:A3871 = AUS, 3: BOASG
         $OUT[3871] = FALSE
      ;ENDFOLD
      ;FOLD -- Dress Fin AUS -- ;%{SE}%MKUKATPVW %CVW_COM %VCOMMENT %P 2:-- Dress Fin AUS --, 3: VW_COMMENT
      ;ENDFOLD
      ;FOLD A3872 = AUS ;%{SE}%MKUKATPVW %CVW_SPS %VBOASG %P 2:A3872 = AUS, 3: BOASG
         $OUT[3872] = FALSE
      ;ENDFOLD
      ;FOLD -- Start StartAcknowledge AUS -- ;%{SE}%MKUKATPVW %CVW_COM %VCOMMENT %P 2:-- Start StartAcknowledge AUS --, 3: VW_COMMENT
      ;ENDFOLD
      ;FOLD A3512 = AUS ;%{SE}%MKUKATPVW %CVW_SPS %VBOASG %P 2:A3512 = AUS, 3: BOASG
         $OUT[3512] = FALSE
      ;ENDFOLD
      ;FOLD -- RSK Sammelstoerung -- ;%{SE}%MKUKATPVW %CVW_COM %VCOMMENT %P 2:-- RSK Sammelstoerung --, 3: VW_COMMENT
      ;ENDFOLD
      ;FOLD F329 = F122 ;%{SE}%MKUKATPVW %CVW_SPS %VBOASG %P 2:F329 = F122, 3: BOASG
         $FLAG[329] = $FLAG[122]
      ;ENDFOLD
      ;FOLD F93 = (!E786 & E787 & !E788 & !F830) + F122 & (E26 + E27) ;%{SE}%MKUKATPVW %CVW_SPS %VBOASG %P 2:F93 = (!E786 & E787 & !E788 & !F830) + F122 & (E26 + E27), 3: BOASG
         $FLAG[93] = (NOT $IN[786] AND $IN[787] AND NOT $IN[788] AND NOT $FLAG[830]) OR $FLAG[122] AND ($IN[26] OR $IN[27])
      ;ENDFOLD
      ;FOLD Schritt 1 = F93 & A4039 & A3862 & A3506 & A3505 ;%{SE}%MKUKATPVW %CVW_SPS %VST_CON %P 2:Schritt 1 = F93 & A4039 & A3862 & A3506 & A3505, 3: ST_CON
         IF $FLAG[93] AND $OUT[4039] AND $OUT[3862] AND $OUT[3506] AND $OUT[3505] THEN
            PREV_STEP[9] = APP_INT_STEP[9]
            APP_INT_STEP[9] = 1
         ENDIF
      ;ENDFOLD
   ;ENDFOLD
   ;FOLD SCHRITT 150 -- st. RZ1 # Fehler Fraesen -- ;%{P}%MKUKATPVW,%CSTEP,%VST_NR,%P 1:SCHRITT, 2:150, 3: st. RZ1 # Fehler Fraesen
      ;FOLD ;%{H}
         Case 150
      ;ENDFOLD
      ;FOLD -- Ausblasen AUS -- ;%{SE}%MKUKATPVW %CVW_COM %VCOMMENT %P 2:-- Ausblasen AUS --, 3: VW_COMMENT
      ;ENDFOLD
      ;FOLD A836 = AUS ;%{SE}%MKUKATPVW %CVW_SPS %VBOASG %P 2:A836 = AUS, 3: BOASG
         $OUT[836] = FALSE
      ;ENDFOLD
      ;FOLD -- Fraesen AUS -- ;%{SE}%MKUKATPVW %CVW_COM %VCOMMENT %P 2:-- Fraesen AUS --, 3: VW_COMMENT
      ;ENDFOLD
      ;FOLD A834 = AUS ;%{SE}%MKUKATPVW %CVW_SPS %VBOASG %P 2:A834 = AUS, 3: BOASG
         $OUT[834] = FALSE
      ;ENDFOLD
      ;FOLD -- Fehler Reset EIN -- ;%{SE}%MKUKATPVW %CVW_COM %VCOMMENT %P 2:-- Fehler Reset EIN --, 3: VW_COMMENT
      ;ENDFOLD
      ;FOLD A3857 = EIN ;%{SE}%MKUKATPVW %CVW_SPS %VBOASG %P 2:A3857 = EIN, 3: BOASG
         $OUT[3857] = TRUE
      ;ENDFOLD
      ;FOLD -- Dress in Position AUS -- ;%{SE}%MKUKATPVW %CVW_COM %VCOMMENT %P 2:-- Dress in Position AUS --, 3: VW_COMMENT
      ;ENDFOLD
      ;FOLD A3871 = AUS ;%{SE}%MKUKATPVW %CVW_SPS %VBOASG %P 2:A3871 = AUS, 3: BOASG
         $OUT[3871] = FALSE
      ;ENDFOLD
      ;FOLD -- Start Dress Fin AUS -- ;%{SE}%MKUKATPVW %CVW_COM %VCOMMENT %P 2:-- Start Dress Fin AUS --, 3: VW_COMMENT
      ;ENDFOLD
      ;FOLD A3872 = AUS ;%{SE}%MKUKATPVW %CVW_SPS %VBOASG %P 2:A3872 = AUS, 3: BOASG
         $OUT[3872] = FALSE
      ;ENDFOLD
      ;FOLD -- Fehler An SPS EIN -- ;%{SE}%MKUKATPVW %CVW_COM %VCOMMENT %P 2:-- Fehler An SPS EIN --, 3: VW_COMMENT
      ;ENDFOLD
      ;FOLD A140 = EIN ;%{SE}%MKUKATPVW %CVW_SPS %VBOASG %P 2:A140 = EIN, 3: BOASG
         $OUT[140] = TRUE
      ;ENDFOLD
      ;FOLD -- Anwahl Zange 1 EIN -- ;%{SE}%MKUKATPVW %CVW_COM %VCOMMENT %P 2:-- Anwahl Zange 1 EIN --, 3: VW_COMMENT
      ;ENDFOLD
      ;FOLD A3858 = EIN ;%{SE}%MKUKATPVW %CVW_SPS %VBOASG %P 2:A3858 = EIN, 3: BOASG
         $OUT[3858] = TRUE
      ;ENDFOLD
      ;FOLD A3533 = EIN ;%{SE}%MKUKATPVW %CVW_SPS %VBOASG %P 2:A3533 = EIN, 3: BOASG
         $OUT[3533] = TRUE
      ;ENDFOLD
      ;FOLD -- Ueberwachungszeit Fehler Fraesen -- ;%{SE}%MKUKATPVW %CVW_COM %VCOMMENT %P 2:-- Ueberwachungszeit Fehler Fraesen --, 3: VW_COMMENT
      ;ENDFOLD
      ;FOLD t11 ( EIN ) = STOP ;%{SE}%MKUKATPVW %CVW_SPS %VTSTOP %P 2:t11 ( EIN ) = STOP, 3: TSTOP
         VW(#SET_TIME,TRUE,11,1,0)
      ;ENDFOLD
